# B&R Automation Studio project vibratorControlWithCurrentController (part 17)

```iecst
		0:
			IF this.responseStructMini.itemNo > 0 OR gMachineInterface.status.machineNotInProduction THEN // only start server when we are about to request images.
				brdkRESTServer_1.enable := TRUE;
				brdkRESTServer_1.pName := ADR('imageMini');
				brdkRESTServer_1.protocol := BRDK_REST_HTTP;
				brdkRESTServer_1.responseContentType := BRDK_REST_HTML;
				serverMini := 10;
			END_IF

		10:
			IF this.responseStructMini.image <> '' THEN
				brdkRESTServer_1.pResponseBody := ADR(this.responseStructMini.image);
				brdkRESTServer_1.responseBodyLength := SIZEOF(this.responseStructMini.image);
				brdkRESTServer_1.responseAction := BRDK_REST_200_OK;
			END_IF

			IF brdkRESTServer_1.status = ERR_OK THEN

			ELSIF brdkRESTServer_1.status <> ERR_FUB_BUSY THEN
				serverStatusError := brdkRESTServer_0.status;
				serverMini := 222;
			END_IF

		222:
			brdkRESTServer_1.enable := FALSE;
			this.TON_0.IN := TRUE;
			this.TON_0.PT := T#500ms;
			this.TON_0();

			IF this.TON_0.Q THEN
				this.TON_0.IN := FALSE;
				this.TON_0();

				serverMini := 0;
			END_IF

	END_CASE

	brdkRESTServer_1();

END_PROGRAM

PROGRAM _EXIT

	brdkRESTClient_0(enable := FALSE);
	brdkRESTServer_0(enable := FALSE);
END_PROGRAM
```

#### local.typ - Local data types
```iecst
TYPE
	local_typ : 	STRUCT
		strURL : STRING[300];
		oldItemNumber : STRING[20];
		errorCode : UINT;
		responeStruct : responeStruct_typ; (*JSON response will be parsed into this structure*)
		responseStructMini : responeStruct_typ;
		TON_0 : TON;
		imageURL : STRING[60];
		tmpStr : STRING[20];
		countPictureChanged : UDINT;
		tmpImageURL : STRING[60];
		TON_client : TON;
		errorCount : USINT;
	END_STRUCT;
	responeStruct_typ : 	STRUCT
		itemNo : DINT;
		image : STRING[99999];
	END_STRUCT;
END_TYPE
```

#### local.var - Local variables
```iecst
VAR
	brdkRESTClient_0 : brdkRESTClient;
	brdkRESTServer_0 : brdkRESTServer;
	requestBody : STRING[99];
	responseBody : STRING[99999];
	this : local_typ;
	state : USINT;
	serverState : USINT;
	message1 : DINT;
	message2 : DINT;
	pictureReady : BOOL;
	serverStatusError : UINT;
	strURL1 : STRING[80] := 'https://ip.uat.cz.pac.corp.lego.com/';
	strURL2 : STRING[80] := 'image-service/api/itemimage/getitemimagedata/';
	image : STRING[99999];
	testImg : USINT;
	oldTestImg : USINT;
	oldNumBricksInPortion : UDINT;
	item : STRING[80];
	quantity : STRING[99];
	serverMini : USINT;
	brdkRESTServer_1 : brdkRESTServer;
END_VAR
```

### Program Logical/services/EthernetIP/ethIp (IEC)

#### Variables.var
```iecst
VAR
	EIPInit_0 : EIPInit;
	EIPCyclic_0 : EIPCyclic;
	EIPExit_0 : EIPExit;
	remoteOutputArray : DINT;
	remoteInputArray : DINT;
	remoteCommectionStatus : UDINT;
	state : USINT;
	tmpStr : STRING[20];
	strInternalLineIP : STRING[20];
	ident : {REDUND_UNREPLICABLE} UDINT;
	ipLineController : STRING[15] := '192.168.1.10';
	interface : REFERENCE TO gEthernetIPInterface_typ;
END_VAR
```

#### Main.st
```iecst
PROGRAM _INIT

	EIPInit_0.enable := TRUE;
	EIPInit_0.pconfig := ADR('eipconf');
	EIPInit_0();

	remoteInputArray;
	remoteOutputArray;
	remoteCommectionStatus;
END_PROGRAM

PROGRAM _CYCLIC

	CASE state OF

		0:
			IF gMachineInterface.parameter.actualServerIP <> '' THEN

				tmpStr := '';
				brdkStrSubStr(ADR(tmpStr),ADR(gMachineInterface.parameter.actualServerIP),-1,3);
				strInternalLineIP := '192.168.1.';
				strInternalLineIP := CONCAT(strInternalLineIP,tmpStr);

				EIPCyclic_0.handle := EIPInit_0.handle;
				EIPCyclic_0.enable := TRUE;
				state := 10;
			END_IF

		10:
			interface ACCESS ADR(gEthernetIPInterface);

			remoteOutputArray.0  := interface.status.stop;
			remoteOutputArray.1  := interface.status.start;
			remoteOutputArray.2	 := interface.status.empty;
			remoteOutputArray.3  := interface.status.emptyMode;
			remoteOutputArray.4  := interface.status.bypassCassette;
			remoteOutputArray.13 := interface.status.di_cassetteReady;
			remoteOutputArray.14 := interface.status.di_cassetteQueue;
			remoteOutputArray.15 := interface.status.do_cassetteRelease;

			EIPCyclic_0();

			gMainInterface.cmd.stopEthIP := remoteInputArray.0;
			gMainInterface.cmd.startEthIP := remoteInputArray.1;
			gMainInterface.cmd.emptyEthIP := remoteInputArray.2;
			gMainInterface.cmd.emptyModeEthIP := remoteInputArray.3;
			gMainInterface.cmd.bypassCassetteEthIP := remoteInputArray.4;

	END_CASE

END_PROGRAM

PROGRAM _EXIT

	EIPExit_0.handle := EIPCyclic_0.handle;
	EIPExit_0.enable := TRUE;
	EIPExit_0();

END_PROGRAM
```

### Data object Logical/services/EthernetIP/eipconf (Simple)

#### DataObject.dat
```
"#OWNINTERFACE=SS1.IF1.ETH"
"#STATION=ROCKWELL"
"#STATIONIP=192.168.1.10"
"#STATIONSTATUS=::ethIp:remoteCommectionStatus"				; Number of active ethernet/IP connections.
"#CONNAME=EIPCon"
"#CONDIR=BOTH"
"#CONRPI=20"														; 20ms interval for requested packet. Need to call EIP FBs at least 2 times as fast as this time!
"#INPUTASSEMBLY=AssemIn"											; From AB side. This data is read by AB from B&R
"::ethIp:remoteOutputArray, DINT, 1"
"#OUTPUTASSEMBLY=AssemOut"											; From AB side. This data is read by B&R from AB
"::ethIp:remoteInputArray, DINT, 1"
```

### global.typ
```iecst
TYPE
	gEthernetIPInterface_typ : 	STRUCT
		status : gEthernetIPInterface_status_typ;
	END_STRUCT;
	gEthernetIPInterface_status_typ : 	STRUCT
		stop : BOOL; (*CM20 to LineController status*)
		start : BOOL; (*CM20 to LineController status*)
		empty : BOOL; (*CM20 to LineController status*)
		emptyMode : BOOL; (*CM20 to LineController status*)
		bypassCassette : BOOL; (*CM20 to LineController status*)
		di_cassetteReady : BOOL;
		di_cassetteQueue : BOOL;
		do_cassetteRelease : BOOL;
	END_STRUCT;
END_TYPE
```

### global.var
```iecst
VAR
	gEthernetIPInterface : gEthernetIPInterface_typ;
END_VAR
```

### dataGlobal.typ - Global data types
```iecst
TYPE
	gData_typ : 	STRUCT  (*Global recipe type.*)
		cmd : gData_cmd_typ; (*Command type.*)
		status : gData_status_typ; (*Status type.*)
	END_STRUCT;
	gData_cmd_typ : 	STRUCT  (*Global command type.*)
		numberOfSamples : UDINT := 250;
		triggerRecord : BOOL;
		exportRecord : BOOL;
		humanDecision : BOOL;
		machineDecision : BOOL;
		startRecord : BOOL;
		enable : BOOL;
	END_STRUCT;
	gData_status_typ : 	STRUCT  (*Global status type.*)
		running : BOOL := TRUE;
		active : BOOL;
		enoughFreeMem : BOOL; (*Will be false if we have less than 10 MiB freemem*)
	END_STRUCT;
END_TYPE
```

### dataGlobal.var - Global variables
```iecst
VAR
	gData : gData_typ; (*Global recipe interface.*)
END_VAR
```

### Package Logical/services/FAT - This module is used to handle all file devices.

### fatGlobal.typ - Global data types
```iecst
TYPE
	gFAT_typ : 	STRUCT  (*Global file type.*)
		cmd : gFAT_cmd_typ; (*File command type.*)
		status : gFAT_status_typ; (*File status type.*)
	END_STRUCT;
	gFAT_status_typ : 	STRUCT  (*File status type.*)
		dummy : BOOL; (*File devices are ready to use.*)
	END_STRUCT;
	gFAT_cmd_typ : 	STRUCT  (*File command type.*)
		dummy : BOOL; (*Update file devices command.*)
	END_STRUCT;
END_TYPE
```

### fatGlobal.var - Global variables
```iecst
VAR
	gFAT : gFAT_typ; (*Global file interface.*)
END_VAR
```

### Program Logical/services/FAT/FAT (IEC, version 1.00.0) - file device management task

#### local.st - Init, cyclic, exit code
```iecst
PROGRAM _INIT

	ST_name(0,ADR(this.configName),0);
	brdkStrCat(ADR(this.configName),ADR(':this.config'));
	ST_name(0,ADR(this.resultName),0);
	brdkStrCat(ADR(this.resultName),ADR(':resultFAT'));

	MpRecipeRegPar_Config.Enable := TRUE;
	this.MpRecipeXml_0.Load := TRUE;
	this.ton_chekForChanges.PT := T#5s;

END_PROGRAM

PROGRAM _CYCLIC

	// If machine aborts stop all tests.
	IF gMainInterface.status.state = STATE_ABORTED THEN
		this.hmi.testRunning88h := this.hmi.testRunning12h := FALSE;
	END_IF

	CASE state OF

		0:
			IF gFile.status.ready AND (gConfig.status.saved OR gConfig.status.loaded) AND this.resultsFATLoaded  THEN

				this.config.timeLeft88h := 88.0-(this.config.timeElapsed88h/3600);
				this.config.timeLeft88h := getHourMinutsFromDecimal(this.config.timeLeft88h);
				this.config.timeLeft12h := 12.0-(this.config.timeElapsed12h/3600);
				this.config.timeLeft12h := getHourMinutsFromDecimal(this.config.timeLeft12h);
				this.hmi.cmd.enableArrowNext := this.hmi.cmd.enableMenuNavigation := resultFAT.initialGroundMeas.done;

				state := 5;

			END_IF

		5:
			IF this.hmi.cmd.startFAT THEN
				// Only go to these states if FAT have been opened
				IF stateRetain > 0 THEN
					state := stateRetain;
				ELSE
					state := 10;
				END_IF
			END_IF

		10:
			// Initial ground measurements

			resultFAT.initialGroundMeas.firstMeasurementDone := resultFAT.initialGroundMeas.measurementValue <= 0.1 AND resultFAT.initialGroundMeas.measurementValue > 0.0;

			resultFAT.resistanceMeas2.done := TRUE;
			FOR i:=0 TO 9 DO

				CASE i OF

					0,1,2,3,7,8:	// 10ohm max resistance.
						IF resultFAT.resistanceMeas2.measurementArr[i]=0.0 OR resultFAT.resistanceMeas2.measurementArr[i] > 0.10 THEN
							resultFAT.resistanceMeas2.done := FALSE;
							resultFAT.resistanceMeas2.measurementOK[i] := FALSE;
						ELSE
							resultFAT.resistanceMeas2.measurementOK[i] := TRUE;
						END_IF

					4,5,6:		// 0.33ohm max resistance.
						IF resultFAT.resistanceMeas2.measurementArr[i]=0.0 OR resultFAT.resistanceMeas2.measurementArr[i] > 0.33 THEN
							resultFAT.resistanceMeas2.done := FALSE;
							resultFAT.resistanceMeas2.measurementOK[i] := FALSE;
						ELSE
							resultFAT.resistanceMeas2.measurementOK[i] := TRUE;
						END_IF

				END_CASE
			END_FOR

			resultFAT.initialGroundMeas.done := resultFAT.initialGroundMeas.firstMeasurementDone AND resultFAT.resistanceMeas2.done;

			this.hmi.cmd.enableArrowNext := this.hmi.cmd.enableMenuNavigation := resultFAT.initialGroundMeas.done;

			IF this.hmi.cmd.arrowNextValue THEN
				this.hmi.cmd.arrowNextValue := FALSE;
				IF resultFAT.initialGroundMeas.done THEN // only continue if it's done.
					state := 20;
				END_IF
			END_IF

		20:
			// Machine setup

			// On edgepos of input disable the oppsite (only 1 of 2 is valid)
			// A lot of information is depending on the machine type. All this information will be used at later steps in the FAT.
			IF EDGEPOS(this.hmi.cmd.smallCfToggleButton) THEN
				this.hmi.cmd.bigCfToggleButton := FALSE;
				gVibratorInterface[0].parameter.CFType := 0;
				gVibratorInterface[0].cmd.setCfType := TRUE;
				resultFAT.machineSetup.strCfSize := 'CM20 small';
				resultFAT.machineSetup.strMaxSpecsCF := 'MAX (2A/200V)';
				resultFAT.additionalInfo.weightOfCf := '5.5kg';
				resultFAT.CFSpringAdjust.strTargetFrequency := '48 - 51';
				resultFAT.CFCoilAdjust.magneticGap := 1.2;
				resultFAT.LFCoilAdjust.magneticGap := 0.6;
				resultFAT.machineSetup.cfSize := 0;
			ELSIF EDGEPOS(this.hmi.cmd.bigCfToggleButton) THEN
				this.hmi.cmd.smallCfToggleButton := FALSE;
				gVibratorInterface[0].parameter.CFType := 1;
				gVibratorInterface[0].cmd.setCfType := TRUE;
				resultFAT.machineSetup.strCfSize := 'CM20 large';
				resultFAT.machineSetup.strMaxSpecsCF := 'MAX (2A/200V)';
				resultFAT.additionalInfo.weightOfCf := '13.5kg';
				resultFAT.CFSpringAdjust.strTargetFrequency := '23.7 - 25.5';
				resultFAT.CFCoilAdjust.magneticGap := 2.5;
				resultFAT.LFCoilAdjust.magneticGap := 0.5;
				resultFAT.machineSetup.cfSize := 1;
			ELSIF EDGEPOS(this.hmi.cmd.leftDirectionOfRotation) THEN
				// direction should be 1 on left machine
				this.hmi.cmd.rightDirectionOfRotation := FALSE;
				gBeltInterface.cmd.setDirection := TRUE;
				gBeltInterface.parameter.direction := 1;
				resultFAT.machineSetup.strMachineType := 'Right';		// A machine with "left direction of rotation" is a right machine.
				resultFAT.machineSetup.strIsItALeftMachine := 'X (Left direction)';
				resultFAT.machineSetup.strIsItARightMachine := '';
				resultFAT.machineSetup.machineType := 0;	// left machine
				//config.machineType := 1;
			ELSIF EDGEPOS(this.hmi.cmd.rightDirectionOfRotation) THEN
				// direction should be 0 on right machine.
				this.hmi.cmd.leftDirectionOfRotation := FALSE;
				gBeltInterface.cmd.setDirection := TRUE;
				gBeltInterface.parameter.direction := 0;
				resultFAT.machineSetup.strMachineType := 'Left';		// A machine with "Right direction of rotation" is a left machine.
				resultFAT.machineSetup.strIsItALeftMachine := '';
				resultFAT.machineSetup.strIsItARightMachine := 'X (Right direction)';
				resultFAT.machineSetup.machineType := 1;	// right machine
				//config.machineType := 0;
			END_IF

			IF resultFAT.machineSetup.done THEN	// in order to load "this.hmi" if machine is restarted. They are not remanent.
				this.hmi.cmd.rightDirectionOfRotation := resultFAT.machineSetup.machineType=1;
				this.hmi.cmd.leftDirectionOfRotation := resultFAT.machineSetup.machineType=0;
				this.hmi.cmd.smallCfToggleButton := resultFAT.machineSetup.cfSize=0;
				this.hmi.cmd.bigCfToggleButton := resultFAT.machineSetup.cfSize=1;
			END_IF

			// Allow user to continue ONLY if their input is valid
			IF (this.hmi.cmd.smallCfToggleButton XOR this.hmi.cmd.bigCfToggleButton) AND
				(this.hmi.cmd.leftDirectionOfRotation XOR this.hmi.cmd.rightDirectionOfRotation) THEN
				resultFAT.machineSetup.done := TRUE;
				this.hmi.cmd.enableArrowNext := TRUE;
			ELSE
				resultFAT.machineSetup.done := FALSE;
				this.hmi.cmd.enableArrowNext := FALSE;
			END_IF

			// COMMENT OUT - this string anyways make 0 sense for report today?
//			IF EDGENEG(gVibratorInterface[0].cmd.setCfType) THEN	// a negative edge means it's done creating the string in vibrator task.
//				resultFAT.machineSetup.strLinearizationAccValuesCF := gVibratorInterface[0].status.strLinearizationAccValues;	// CF string
//				resultFAT.machineSetup.strLinearizationAccValuesLF := gVibratorInterface[1].status.strLinearizationAccValues;	// LF string
//			END_IF

			// User input to continue to next step
			IF this.hmi.cmd.arrowNextValue THEN
				this.hmi.cmd.arrowNextValue := FALSE;	// reset.

				// Set vibrator unit type and "top unit type" auto
				IF resultFAT.machineSetup.cfSize = 0 AND resultFAT.machineSetup.machineType = 0 THEN	//  small and left
					resultFAT.additionalInfo.vibratorUnitType := 'SRC-N 250-2L-LEGO II';
					resultFAT.additionalInfo.topUnitType := 'PJ 2016 HA';
				ELSIF resultFAT.machineSetup.cfSize = 0 AND resultFAT.machineSetup.machineType = 1 THEN	//  small and right
					resultFAT.additionalInfo.vibratorUnitType := 'SRC-N 250-2R-LEGO II';
					resultFAT.additionalInfo.topUnitType := 'PJ 2016 VA';
				ELSIF resultFAT.machineSetup.cfSize = 1 AND resultFAT.machineSetup.machineType = 0 THEN	//  big and left
					resultFAT.additionalInfo.vibratorUnitType := 'SRC-N 400-1L-LEGO III';
					resultFAT.additionalInfo.topUnitType := 'PJ 99 HA';
				ELSIF resultFAT.machineSetup.cfSize = 1 AND resultFAT.machineSetup.machineType = 1 THEN	//  big and right
					resultFAT.additionalInfo.vibratorUnitType := 'SRC-N 400-1R-LEGO III';
					resultFAT.additionalInfo.topUnitType := 'PJ 99 VA';
				END_IF

				state := 30;
			ELSIF this.hmi.cmd.arrowBackValue THEN
				this.hmi.cmd.arrowBackValue := FALSE;
				state := 10;
			END_IF

		30:
			// Wing connector (wingTestIO)

			IF this.hmi.cmd.arrowNextValue THEN			// go to next
				this.hmi.cmd.arrowNextValue := FALSE;	// reset
				state := 40;
			ELSIF this.hmi.cmd.arrowBackValue THEN
				this.hmi.cmd.arrowBackValue := FALSE;
				state := 20;
			END_IF

		40:
			// Additional machine info

			// Create string typeNo.-SerialNo.
			IF resultFAT.additionalInfo.serialNo <> '' AND resultFAT.additionalInfo.typeNo <> '' THEN
				brdkStrMemSet(ADR(resultFAT.additionalInfo.typeNoAndSerialNo),0,SIZEOF(resultFAT.additionalInfo.typeNoAndSerialNo));
				brdkStrCat(ADR(resultFAT.additionalInfo.typeNoAndSerialNo),ADR(resultFAT.additionalInfo.typeNo));
				this.tmpString := '-';
				brdkStrCat(ADR(resultFAT.additionalInfo.typeNoAndSerialNo),ADR(this.tmpString));
				brdkStrCat(ADR(resultFAT.additionalInfo.typeNoAndSerialNo),ADR(resultFAT.additionalInfo.serialNo));

				// SerialNoDINT
				this.tmpString := '';
				brdkStrCat(ADR(this.tmpString),ADR(resultFAT.additionalInfo.typeNo));
				brdkStrCat(ADR(this.tmpString),ADR(resultFAT.additionalInfo.serialNo));
				gMachineInterface.cmd.serialNoDINT := STRING_TO_DINT(this.tmpString); //interface.par.serialNoDINT := STRING_TO_DINT(this.tmpString);
			END_IF
			//interface.par.serialNo := resultFAT.additionalInfo.typeNoAndSerialNo;

			// Load "this.hmi.status" texts if they are empty and resultFAT is not (Happens on a warm restart).
			IF this.hmi.status.additionalInfo.typeNo = 0 AND resultFAT.additionalInfo.typeNo <> '' THEN
				this.hmi.status.additionalInfo.typeNo := STRING_TO_UDINT(resultFAT.additionalInfo.typeNo);
			END_IF
			IF this.hmi.status.additionalInfo.serialNo = 0 AND resultFAT.additionalInfo.serialNo <> '' THEN
				this.hmi.status.additionalInfo.serialNo := STRING_TO_UDINT(resultFAT.additionalInfo.serialNo);
			END_IF
			IF this.hmi.status.additionalInfo.rnoNo = 0.0 AND resultFAT.additionalInfo.rnaProductNo <> '' THEN
				this.hmi.status.additionalInfo.rnoNo := STRING_TO_LREAL(resultFAT.additionalInfo.rnaProductNo);
			END_IF
			IF this.hmi.status.additionalInfo.topSerialNo = 0 AND resultFAT.additionalInfo.topSerialNo <> '' THEN
				this.hmi.status.additionalInfo.topSerialNo := STRING_TO_UDINT(resultFAT.additionalInfo.topSerialNo);
			END_IF

			// Put int into strings for report
			resultFAT.additionalInfo.typeNo := UDINT_TO_STRING(this.hmi.status.additionalInfo.typeNo);
			resultFAT.additionalInfo.serialNo := UDINT_TO_STRING(this.hmi.status.additionalInfo.serialNo);
			resultFAT.additionalInfo.rnaProductNo := LREAL_TO_STRING(this.hmi.status.additionalInfo.rnoNo);
			resultFAT.additionalInfo.topSerialNo := UDINT_TO_STRING(this.hmi.status.additionalInfo.topSerialNo);

			IF this.hmi.status.additionalInfo.IRTHno <> this.oldLREAL THEN
				resultFAT.additionalInfo.IRTHno := LREAL_TO_STRING(this.hmi.status.additionalInfo.IRTHno);
				brdkStrRemove(ADR(resultFAT.additionalInfo.IRTHno),(brdkStrLen(ADR(resultFAT.additionalInfo.IRTHno))-2),2);

				IF this.hmi.status.additionalInfo.IRTHno>10000000 THEN // hacky way to append a space to a numeric input from HMI.
					this.tmpString := ' ';
					brdkStrInsertAtPos(ADR(resultFAT.additionalInfo.IRTHno),ADR(this.tmpString),6);
				END_IF
			END_IF
			this.oldLREAL := this.hmi.status.additionalInfo.IRTHno;

			IF this.hmi.cmd.arrowNextValue THEN
				this.hmi.cmd.arrowNextValue := FALSE;
				state := 50;
			ELSIF this.hmi.cmd.arrowBackValue THEN
				this.hmi.cmd.arrowBackValue := FALSE;
				state := 30;
			END_IF

			// If some chars in all text inputs the test is done:
			IF resultFAT.additionalInfo.IRTHno <> '0' AND resultFAT.additionalInfo.IRTHno <> '0.0' AND resultFAT.additionalInfo.rnaProductNo <> '0.0' AND resultFAT.additionalInfo.typeNo <> '0' AND resultFAT.additionalInfo.serialNo <> '0' AND resultFAT.additionalInfo.topSerialNo <> '0' AND resultFAT.additionalInfo.topUnitType <> '' AND resultFAT.additionalInfo.vibratorUnitType <> '' THEN
				resultFAT.additionalInfo.done := TRUE;
			ELSE
				resultFAT.additionalInfo.done := FALSE;
			END_IF

		50:

			//Capcon voltage measurement

			// Check if user input is in the expected interval
			IF resultFAT.capconMeasurement.V1 >= 18 - this.maxPlusMinusVoltage AND resultFAT.capconMeasurement.V1 <= 18 + this.maxPlusMinusVoltage THEN
				this.hmi.cmd.crossmarkV1 := 1;
			ELSE
				this.hmi.cmd.crossmarkV1 := 0;
			END_IF

			// Check if user input is in the expected interval
			IF resultFAT.capconMeasurement.V2 >= -15.8 - this.maxPlusMinusVoltage AND resultFAT.capconMeasurement.V2 <= -15.8 + this.maxPlusMinusVoltage THEN
				this.hmi.cmd.crossmarkV2 := 1;
			ELSE
				this.hmi.cmd.crossmarkV2 := 0;
			END_IF

			IF (this.hmi.cmd.crossmarkV1 > 0 AND this.hmi.cmd.crossmarkV2 > 0) THEN
				resultFAT.capconMeasurement.done := TRUE;
				this.hmi.cmd.enableArrowNext := TRUE;
			ELSE
				resultFAT.capconMeasurement.done := FALSE;
				this.hmi.cmd.enableArrowNext := FALSE;
			END_IF

			IF this.hmi.cmd.arrowNextValue THEN
				this.hmi.cmd.arrowNextValue := FALSE;
				state := 60;
			ELSIF this.hmi.cmd.arrowBackValue THEN
				this.hmi.cmd.arrowBackValue := FALSE;
				state := 40;
			END_IF

		60:
			//	em.description := 'Capcon signal test';
			// 1st test. Test that an analog input is getting into the machine when dropping something through capcon:

			// 2nd test. Auto test MAX speed signal doing a period of 5s.
			IF EDGEPOS(this.hmi.cmd.startCapconTest2) THEN
				gCapconInterface.status.maxRawSignal := 0;
				gCapconInterface.cmd.startSpeedSignalTest := TRUE;
			END_IF

			IF EDGENEG(gCapconInterface.cmd.startSpeedSignalTest) THEN
				this.hmi.cmd.startCapconTest2 := FALSE;
				this.hmi.status.maxRawSignal := ABS(gCapconInterface.status.maxRawSignal);
				IF this.hmi.status.maxRawSignal>1 AND ABS(this.hmi.status.maxRawSignal) < 100 THEN // TODO: 40 NEEDS TO BE TESTED!
					resultFAT.capconTest.signalTest2 := TRUE;
				ELSE
					resultFAT.capconTest.signalTest2 := FALSE;
				END_IF
			END_IF

			IF this.hmi.cmd.arrowNextValue THEN
				this.hmi.cmd.arrowNextValue := FALSE;
				state := 70;
			ELSIF this.hmi.cmd.arrowBackValue THEN
				this.hmi.cmd.arrowBackValue := FALSE;
				state := 50;
			END_IF

			resultFAT.capconTest.done := resultFAT.capconTest.signalTest1 AND resultFAT.capconTest.signalTest2;

		70:
			// em.description := 'Level sensor test';

			gFeederInterface.cmd.levelSensorTestActive := TRUE;

			IF this.hmi.cmd.doLevelSensorTest AND resultFAT.levelSensorTest.receiverOK THEN

				// level sensor test.
				CASE levelTestState OF

					0:
						gFeederInterface.cmd.setLevelSensor[0] := FALSE;
						gFeederInterface.cmd.setLevelSensor[1] := FALSE;
						gFeederInterface.cmd.setLevelSensor[2] := TRUE;
						resultFAT.levelSensorTest.transmitterLowOK := FALSE;
						resultFAT.levelSensorTest.transmitterMediumOK := FALSE;
						resultFAT.levelSensorTest.transmitterHighOK := FALSE;
						resultFAT.levelSensorTest.operatorApproveLow := resultFAT.levelSensorTest.operatorApproveMedium := resultFAT.levelSensorTest.operatorApproveHigh := FALSE;

						this.timeElapsed := 0;
						levelTestState := 5;

					5:	// wait 1s
						this.timeElapsed := this.timeElapsed + 40000;
						IF this.timeElapsed > 1000000 THEN
							this.timeElapsed := 0;
							IF gFeederInterface.status.levelSensorReceiverInBowl THEN
								levelTestState := 222;
							ELSE
								this.hmi.status.styleToggleInputHigh := TRUE;
								levelTestState := 10;
							END_IF
						END_IF

					10: // Wait for user to approve that HIGH transmitter is flashing.

						IF gFeederInterface.status.levelSensorReceiverInBowl THEN
							levelTestState := 222;
						ELSIF resultFAT.levelSensorTest.operatorApproveHigh THEN
							resultFAT.levelSensorTest.transmitterHighOK := TRUE;

							gFeederInterface.cmd.setLevelSensor[0] := FALSE;
							gFeederInterface.cmd.setLevelSensor[1] := TRUE;
							gFeederInterface.cmd.setLevelSensor[2] := FALSE;
							this.hmi.status.styleToggleInputHigh := FALSE;
							this.hmi.status.styleToggleInputMedium := TRUE;
							levelTestState := 20;
						END_IF

					20: // Wait for user to approve that MEDIUM transmitter is flashing.

						IF gFeederInterface.status.levelSensorReceiverInBowl THEN
							levelTestState := 222;
						ELSIF resultFAT.levelSensorTest.operatorApproveMedium THEN
							resultFAT.levelSensorTest.transmitterMediumOK := TRUE;

							gFeederInterface.cmd.setLevelSensor[0] := TRUE;
							gFeederInterface.cmd.setLevelSensor[1] := FALSE;
							gFeederInterface.cmd.setLevelSensor[2] := FALSE;
							this.hmi.status.styleToggleInputMedium := FALSE;
							this.hmi.status.styleToggleInputLow := TRUE;

							levelTestState := 30;
						END_IF

					30: //  Wait for user to approve that LOW transmitter is flashing.

						IF gFeederInterface.status.levelSensorReceiverInBowl THEN
							levelTestState := 222;
						ELSIF resultFAT.levelSensorTest.operatorApproveLow THEN
							resultFAT.levelSensorTest.transmitterLowOK := TRUE;

							gFeederInterface.cmd.setLevelSensor[0] := FALSE;
							gFeederInterface.cmd.setLevelSensor[1] := FALSE;
							gFeederInterface.cmd.setLevelSensor[2] := FALSE;
							this.hmi.status.styleToggleInputLow := FALSE;
							this.hmi.cmd.doLevelSensorTest := FALSE;
							levelTestState := 0;
						END_IF

					222:
						//test failed reset everything
						this.hmi.cmd.doLevelSensorTest := FALSE;
						gFeederInterface.cmd.setLevelSensor[0] := FALSE;
						gFeederInterface.cmd.setLevelSensor[1] := FALSE;
						gFeederInterface.cmd.setLevelSensor[2] := FALSE;
						resultFAT.levelSensorTest.operatorApproveHigh := resultFAT.levelSensorTest.operatorApproveMedium := resultFAT.levelSensorTest.operatorApproveLow := FALSE;
						resultFAT.levelSensorTest.transmitterLowOK := FALSE;
						resultFAT.levelSensorTest.transmitterMediumOK := FALSE;
						resultFAT.levelSensorTest.transmitterHighOK := FALSE;
						this.hmi.status.styleToggleInputHigh := this.hmi.status.styleToggleInputMedium := this.hmi.status.styleToggleInputLow := FALSE;
						levelTestState := 0;

				END_CASE

			ELSIF this.hmi.cmd.doLevelSensorTest THEN
				this.hmi.cmd.doLevelSensorTest := FALSE; // reset if user presses button when receiver is not OK.
			ELSE
				// manuel control from user.
				gFeederInterface.cmd.setLevelSensor[0] := this.hmi.cmd.setLevelSensorLow;
				gFeederInterface.cmd.setLevelSensor[1] := this.hmi.cmd.setLevelSensorMedium;
				gFeederInterface.cmd.setLevelSensor[2] := this.hmi.cmd.setLevelSensorHigh;

				IF NOT this.hmi.cmd.setLevelSensorHigh AND NOT this.hmi.cmd.setLevelSensorMedium AND NOT this.hmi.cmd.setLevelSensorLow THEN
					// if receiver is high when all transmitters are low the receiver is OK.
					IF gFeederInterface.status.levelSensorReceiverInBowl THEN
						resultFAT.levelSensorTest.receiverOK := TRUE;
					ELSE
						resultFAT.levelSensorTest.receiverOK := FALSE;
					END_IF
				END_IF

			END_IF

			IF this.hmi.cmd.arrowNextValue THEN
				this.hmi.cmd.arrowNextValue := FALSE;	// reset.
				gFeederInterface.cmd.levelSensorTestActive := FALSE;
				state := 80;
			ELSIF this.hmi.cmd.arrowBackValue THEN
				this.hmi.cmd.arrowBackValue := FALSE;
				gFeederInterface.cmd.levelSensorTestActive := FALSE;
				state := 60;
			END_IF

			resultFAT.levelSensorTest.done := resultFAT.levelSensorTest.receiverOK AND resultFAT.levelSensorTest.transmitterHighOK AND resultFAT.levelSensorTest.transmitterMediumOK AND resultFAT.levelSensorTest.transmitterLowOK;
			//this.hmi.cmd.enableArrowNext := resultFAT.levelSensorTest.done;

		80:
			//  'Photo sensor adjustment';

			IF this.hmi.cmd.arrowNextValue THEN
				this.hmi.cmd.arrowNextValue := FALSE;	// reset.
				state := 90;
			ELSIF this.hmi.cmd.arrowBackValue THEN
				this.hmi.cmd.arrowBackValue := FALSE;
				state := 70;
			END_IF

			this.hmi.cmd.enableArrowNext := resultFAT.photoSensorAdjust.done;

		90:
		//	em.description := 'Wait for automatic test of photo sensor to be done';

			IF EDGEPOS(this.hmi.cmd.doPhotoSensorTest) THEN		// Start the test.

				this.hmi.status.photoSensorTestText := 0;
				gBeltInterface.cmd.doPhotoSensorTest := TRUE;						// signal to belt that it should start automatic test.
			ELSIF EDGEPOS(this.hmi.cmd.doPhotoSensorTestNoBelt) THEN

				gBeltInterface.cmd.doPhotoSensorTestNoBelt := TRUE;
			ELSE
				IF gBeltInterface.status.photoSensorTestResult = TEST_STOPPED THEN
					resultFAT.photoSensorTest.testWithBelt := FALSE;
					gBeltInterface.status.photoSensorTestResult := TEST_NOT_DONE;
					this.hmi.cmd.doPhotoSensorTest := FALSE;
					this.hmi.status.photoSensorTestText := 3;	// test stopped text
				ELSIF gBeltInterface.status.photoSensorTestResult = TEST_NOT_OK THEN	// Something went wrong doing test.
					resultFAT.photoSensorTest.testWithBelt := FALSE;
					gBeltInterface.status.photoSensorTestResult := TEST_NOT_DONE;
					this.hmi.cmd.doPhotoSensorTest := FALSE;
					this.hmi.status.photoSensorTestText := 2;
				ELSIF gBeltInterface.status.photoSensorTestResult = TEST_OK THEN
					resultFAT.photoSensorTest.testWithBelt := TRUE;
					gBeltInterface.status.photoSensorTestResult := TEST_NOT_DONE;
					this.hmi.cmd.doPhotoSensorTest := FALSE;
					this.hmi.status.photoSensorTestText := 1;
				END_IF

				IF gBeltInterface.status.photoSensorTestNoBeltResult = TEST_STOPPED THEN
					resultFAT.photoSensorTest.testWithNoBelt := FALSE;
					gBeltInterface.status.photoSensorTestNoBeltResult := TEST_NOT_DONE;
					this.hmi.cmd.doPhotoSensorTestNoBelt := FALSE;
				ELSIF gBeltInterface.status.photoSensorTestNoBeltResult = TEST_NOT_OK THEN	// Something went wrong doing test.
					resultFAT.photoSensorTest.testWithNoBelt := FALSE;
					gBeltInterface.status.photoSensorTestNoBeltResult := TEST_NOT_DONE;
					this.hmi.cmd.doPhotoSensorTestNoBelt := FALSE;
				ELSIF gBeltInterface.status.photoSensorTestNoBeltResult = TEST_OK THEN
					resultFAT.photoSensorTest.testWithNoBelt := TRUE;
					gBeltInterface.status.photoSensorTestNoBeltResult := TEST_NOT_DONE;
					this.hmi.cmd.doPhotoSensorTestNoBelt := FALSE;
				END_IF

			END_IF

			IF this.hmi.cmd.arrowNextValue THEN			// go to next
				this.hmi.cmd.arrowNextValue := FALSE;	// reset
				state := 100;
			ELSIF this.hmi.cmd.arrowBackValue THEN
				this.hmi.cmd.arrowBackValue := FALSE;
				state := 80;
			END_IF

			IF resultFAT.photoSensorTest.testWithBelt THEN
				this.hmi.status.photoSensorTestText := 1;
			END_IF
			resultFAT.photoSensorTest.done := resultFAT.photoSensorTest.testWithBelt AND resultFAT.photoSensorTest.testWithNoBelt;
			this.hmi.cmd.enableArrowNext := resultFAT.photoSensorTest.done;

		100:
			// 'Belt feeder test IO - 1';

			IF EDGEPOS(this.hmi.cmd.doBfFlapTest) THEN
				//	this.hmi.cmd.doBfFlapTest := FALSE;		// reset this when test is done instead!!
				// start flap test in feeder task
				resultFAT.bfTestIO.flapTestDone := FALSE;
				gFeederInterface.cmd.startFlapTest := TRUE;
			ELSE
				// reach on test result from flap test.
				IF gFeederInterface.status.flapTest = TEST_STOPPED THEN
					resultFAT.bfTestIO.flapTestDone := FALSE;
					gFeederInterface.status.flapTest := TEST_NOT_DONE;
					this.hmi.cmd.doBfFlapTest := FALSE;
				ELSIF gFeederInterface.status.flapTest = TEST_NOT_OK THEN	// Something went wrong doing test.
					resultFAT.bfTestIO.flapTestDone := FALSE;
					gFeederInterface.status.flapTest := TEST_NOT_DONE;
					this.hmi.cmd.doBfFlapTest := FALSE;
				ELSIF gFeederInterface.status.flapTest = TEST_OK THEN
					resultFAT.bfTestIO.flapTestDone := TRUE;
					gFeederInterface.status.flapTest := TEST_NOT_DONE;
					this.hmi.cmd.doBfFlapTest := FALSE;
				END_IF
			END_IF

			resultFAT.bfTestIO.done := resultFAT.bfTestIO.approveIOsManually AND resultFAT.bfTestIO.approveMainsVoltage AND resultFAT.bfTestIO.flapTestDone;

			IF this.hmi.cmd.arrowNextValue THEN			// go to next
				this.hmi.cmd.arrowNextValue := FALSE;	// reset
				state := 110;
			ELSIF this.hmi.cmd.arrowBackValue THEN
				this.hmi.cmd.arrowBackValue := FALSE;
				state := 90;
			END_IF

		110:
			// 'Wing test IO - flap namur sensor, cassette signal, dosing signal, cassette queue';

			IF EDGEPOS(this.hmi.cmd.doWingTestManuel) THEN
				//this.hmi.cmd.doWingTestManuel := FALSE;
				gUpperFlapInterface.cmd.wingTestManual := TRUE; // Only start upper - they will start each other "sequantially"

				// Reset test results
				resultFAT.wingTestIO.upperFlapOK := FALSE;
				resultFAT.wingTestIO.middleFlapOK := FALSE;
				resultFAT.wingTestIO.bottomFlapOK := FALSE;
				resultFAT.wingTestIO.neighbourFlapOK := FALSE;
				resultFAT.wingTestIO.cassetteReleaseOK := FALSE;
				resultFAT.wingTestIO.ioTestOK := FALSE;

			END_IF

			IF this.hmi.cmd.doWingTestManuel THEN

				// Wait for all tests to be done
				IF NOT gUpperFlapInterface.cmd.wingTestManual AND NOT gMiddleFlapInterface.cmd.wingTestManual AND NOT gBottomFlapInterface.cmd.wingTestManual AND NOT gCassetteInterface.cmd.wingTestManual THEN
					this.hmi.cmd.doWingTestManuel := FALSE;

					// write result from test into resultFAT struct
					resultFAT.wingTestIO.upperFlapOK := gUpperFlapInterface.status.testResultFAT;
					resultFAT.wingTestIO.middleFlapOK := gMiddleFlapInterface.status.testResultFAT;
					resultFAT.wingTestIO.bottomFlapOK := gBottomFlapInterface.status.testResultFAT;
					resultFAT.wingTestIO.neighbourFlapOK := gBottomFlapInterface.status.testResultFAT; // bottom also test neighbour
					resultFAT.wingTestIO.cassetteReleaseOK := gCassetteInterface.status.testResultFAT;
					resultFAT.wingTestIO.ioTestOK := resultFAT.wingTestIO.upperFlapOK AND resultFAT.wingTestIO.middleFlapOK AND resultFAT.wingTestIO.bottomFlapOK AND resultFAT.wingTestIO.neighbourFlapOK AND resultFAT.wingTestIO.cassetteReleaseOK;

				END_IF

			END_IF

			resultFAT.wingTestIO.done := resultFAT.wingTestIO.ioTestOK AND resultFAT.wingTestIO.approveFunctionality;

			IF this.hmi.cmd.arrowNextValue THEN			// go to next
				this.hmi.cmd.arrowNextValue := FALSE;	// reset
				state := 120;
			ELSIF this.hmi.cmd.arrowBackValue THEN
				this.hmi.cmd.arrowBackValue := FALSE;
				state := 100;
			END_IF

		120:
			//	'CF coils adjustments';

			this.hmi.status.isSmallMachine := gVibratorInterface[0].parameter.machineSize=0;
			this.hmi.status.isBigMachine := gVibratorInterface[0].parameter.machineSize=1;

			IF this.hmi.cmd.arrowNextValue THEN
				this.hmi.cmd.arrowNextValue := FALSE;	// reset.
				// Set default amount of plates if all plate values are set to 0 (means no user input).
				FOR i:=0 TO 2 DO
					IF resultFAT.CFSpringAdjust.plate08mm[i] > 0 OR resultFAT.CFSpringAdjust.plate09mm[i] > 0 OR resultFAT.CFSpringAdjust.plate15mm[i] > 0 OR resultFAT.CFSpringAdjust.plate20mm[i] > 0 OR resultFAT.CFSpringAdjust.plate25mm[i] > 0 THEN
						EXIT;
					ELSIF i=2 THEN	// If all all values are 0 set the default amount of plates for this CF.
						IF resultFAT.machineSetup.cfSize=0 THEN // Default for small cf is 5 2.0mm plates on each spring.
							resultFAT.CFSpringAdjust.plate20mm[0] := 5;
							resultFAT.CFSpringAdjust.plate20mm[1] := 5;
							resultFAT.CFSpringAdjust.plate20mm[2] := 5;
						ELSE	// default for big cf is 7 2.0mm plates on each spring
							resultFAT.CFSpringAdjust.plate20mm[0] := 7;
							resultFAT.CFSpringAdjust.plate20mm[1] := 7;
							resultFAT.CFSpringAdjust.plate20mm[2] := 7;
						END_IF
					END_IF

				END_FOR

				state := 130;
			ELSIF this.hmi.cmd.arrowBackValue THEN
				this.hmi.cmd.arrowBackValue := FALSE;
				state := 110;
			END_IF

		130:
			// CF spring adjustments

			IF this.hmi.cmd.startCalibration THEN
				this.hmi.cmd.startCalibration := FALSE;
				// Need to use this bool to differentiate if it was a "FAT calibration" or a "normal calibration".
				gVibratorInterface[0].status.calibratingMode := TRUE;
				this.cfCali := TRUE;
			END_IF

			IF gVibratorInterface[0].status.calibrationResultsReady THEN
				gVibratorInterface[0].status.calibrationResultsReady := FALSE;
				this.hmi.cmd.startCalibration := FALSE;

				IF this.cfCali THEN
					// Take results from calibration and save in resultFAT
					resultFAT.CFSpringAdjust.ressFrequency := gVibratorInterface[0].status.calibrationResultFrequency;
					resultFAT.CFSpringAdjust.maxCurrent := gVibratorInterface[0].status.calibrationResultCurrent;
					resultFAT.CFSpringAdjust.currentOK := gVibratorInterface[0].status.calibrationResultCurrentOK;
					resultFAT.CFSpringAdjust.frequencyOK := gVibratorInterface[0].status.calibrationResultFrequencyOK;
				END_IF
				this.cfCali := FALSE;
			END_IF

			resultFAT.CFSpringAdjust.done := resultFAT.CFSpringAdjust.currentOK AND resultFAT.CFSpringAdjust.frequencyOK;

			IF this.hmi.cmd.arrowNextValue THEN			// go to next
				this.hmi.cmd.arrowNextValue := FALSE;	// reset
				state := 140;
			ELSIF this.hmi.cmd.arrowBackValue THEN
				this.hmi.cmd.arrowBackValue := FALSE;
				state := 120;
			END_IF

		140:
			// 'LF coils adjustment';	// might need to make more substates for CF and LF.

			IF this.hmi.cmd.arrowNextValue THEN
				this.hmi.cmd.arrowNextValue := FALSE;	// reset.
				// Set default amount of plates if all plate values are set to 0 (means no user input).
				FOR i:=0 TO 1 DO
					IF resultFAT.LFSpringAdjust.plate08mm[i] > 0 OR resultFAT.LFSpringAdjust.plate09mm[i] > 0 OR resultFAT.LFSpringAdjust.plate15mm[i] > 0 OR resultFAT.LFSpringAdjust.plate20mm[i] > 0 OR resultFAT.LFSpringAdjust.plate25mm[i] > 0 THEN
						EXIT;
					ELSIF i=1 THEN	// If all all values are 0 set the default amount of plates for this CF.
						IF resultFAT.machineSetup.cfSize=0 THEN // Default for small cm
							resultFAT.LFSpringAdjust.plate08mm[0] := 2;
							resultFAT.LFSpringAdjust.plate08mm[1] := 1;
						ELSE	// default for big cm
							resultFAT.LFSpringAdjust.plate08mm[0] := 1;
							resultFAT.LFSpringAdjust.plate08mm[1] := 1;
							resultFAT.LFSpringAdjust.plate09mm[0] := 1;
						END_IF
					END_IF

				END_FOR

				state := 150;
			ELSIF this.hmi.cmd.arrowBackValue THEN
				this.hmi.cmd.arrowBackValue := FALSE;
				state := 130;
			END_IF

		150:
			// LF calibration

			IF this.hmi.cmd.startCalibration THEN
				this.hmi.cmd.startCalibration := FALSE;
				// Need to use this bool to differentiate if it was a "FAT calibration" or a "normal calibration".
				gVibratorInterface[1].status.calibratingMode := TRUE;
				this.lfCali := TRUE;
			END_IF

			IF gVibratorInterface[1].status.calibrationResultsReady THEN
				gVibratorInterface[1].status.calibrationResultsReady := FALSE;
				this.hmi.cmd.startCalibration := FALSE;

				IF this.lfCali THEN
					// Take results from calibration and save in resultFAT
					resultFAT.LFSpringAdjust.ressFrequency := gVibratorInterface[1].status.calibrationResultFrequency;
					resultFAT.LFSpringAdjust.maxCurrent := gVibratorInterface[1].status.calibrationResultCurrent;
					resultFAT.LFSpringAdjust.currentOK := gVibratorInterface[1].status.calibrationResultCurrentOK;
					resultFAT.LFSpringAdjust.frequencyOK := gVibratorInterface[1].status.calibrationResultFrequencyOK;

					resultFAT.LFSpringAdjust.strResultForReport := REAL_TO_STRING(resultFAT.LFSpringAdjust.maxCurrent);
					resultFAT.LFSpringAdjust.strResultForReport := CONCAT(resultFAT.LFSpringAdjust.strResultForReport,'A');
					resultFAT.LFSpringAdjust.strResultForReport := CONCAT(resultFAT.LFSpringAdjust.strResultForReport,' / ');
					this.tmpString := REAL_TO_STRING(resultFAT.LFSpringAdjust.ressFrequency);
					resultFAT.LFSpringAdjust.strResultForReport := CONCAT(resultFAT.LFSpringAdjust.strResultForReport,this.tmpString);
					resultFAT.LFSpringAdjust.strResultForReport := CONCAT(resultFAT.LFSpringAdjust.strResultForReport,'Hz');

				END_IF
				this.lfCali := FALSE;
			END_IF

			resultFAT.LFSpringAdjust.done := resultFAT.LFSpringAdjust.currentOK AND resultFAT.LFSpringAdjust.frequencyOK;

			IF this.hmi.cmd.arrowNextValue THEN			// go to next
				this.hmi.cmd.arrowNextValue := FALSE;	// reset
				state := 160;
			ELSIF this.hmi.cmd.arrowBackValue THEN
				this.hmi.cmd.arrowBackValue := FALSE;
				state := 140;
			END_IF

		160:
			// 88h test
			this.testRunning := this.hmi.testRunning88h XOR this.hmi.testRunning12h;
			gBeltInterface.cmd.runManualTest := gVibratorInterface[0].cmd.runManualTest := gVibratorInterface[1].cmd.runManualTest := this.testRunning;

			IF this.hmi.testRunning88h AND this.hmi.testRunning12h THEN
				// Both can't run at the same time. Disable both if user tries to do this.
				this.hmi.testRunning88h := this.hmi.testRunning12h := FALSE;
			ELSIF this.hmi.testRunning88h THEN

				// Start belt and vibrators
				gBeltInterface.parameter.speedManualTest := 400.0;
				gVibratorInterface[0].parameter.speedPctManualTest := SEL(this.config.timeElapsed88h > 43200,40.0,80.0); // First 12h use 40% rest of the time use 80% (43200s = 12hours)
				gVibratorInterface[1].parameter.speedPctManualTest := 100.0;

				// Calculate time
				this.config.timeElapsed88h := this.config.timeElapsed88h + CYCLE_TIME_seconds;
				this.config.timeLeft88h := 88.0-(this.config.timeElapsed88h/3600);
				this.config.timeLeft88h := getHourMinutsFromDecimal(this.config.timeLeft88h);

				IF this.config.timeLeft88h <= 0.0 THEN
					this.hmi.testRunning88h := this.hmi.testRunning12h := FALSE;
					gConfig.cmd.save := TRUE;
					this.config.timeLeft88h := 0.0;
					resultFAT.longTest88h.done := TRUE;
				END_IF

			END_IF

			// Save to config every 10min
			this.TON_0.IN := this.testRunning;
			this.TON_0.PT := T#10m;
			this.TON_0();

			IF this.TON_0.Q THEN
				this.TON_0.IN := FALSE;
				this.TON_0();

				gConfig.cmd.save := TRUE;
			END_IF

			// If test not running set parameter to 0.
			IF NOT this.testRunning THEN
				gVibratorInterface[0].parameter.speedPctManualTest := 0.0;
				gVibratorInterface[1].parameter.speedPctManualTest := 0.0;
			END_IF

			IF this.hmi.cmd.arrowNextValue THEN			// go to next
				this.hmi.cmd.arrowNextValue := FALSE;	// reset
				state := 170;
			ELSIF this.hmi.cmd.arrowBackValue THEN
				this.hmi.cmd.arrowBackValue := FALSE;
				state := 150;
			END_IF

		170:
			// 'After 72H test adjustments';

			resultFAT.after72hAdjustments.done := resultFAT.after72hAdjustments.approveCoverMounting AND resultFAT.after72hAdjustments.approveHabasitMounting AND resultFAT.after72hAdjustments.approvePacemakerMarking AND resultFAT.after72hAdjustments.approveRNAmarking;

			IF this.hmi.cmd.arrowNextValue THEN
				this.hmi.cmd.arrowNextValue := FALSE;	// reset.
				state := 180;
			ELSIF this.hmi.cmd.arrowBackValue THEN
				this.hmi.cmd.arrowBackValue := FALSE;
				state := 160;
			END_IF

		180:
			// Calibrate CF again after habasit (LF should not be needed since it has habasit on from the start)

			IF this.hmi.cmd.startCalibration THEN
				this.hmi.cmd.startCalibration := FALSE;
				this.cfCaliHabasit := TRUE; //save what kind of FAT cali which is running.
				gVibratorInterface[0].status.calibratingMode := TRUE;
			END_IF

			IF gVibratorInterface[0].status.calibrationResultsReady THEN
				gVibratorInterface[0].status.calibrationResultsReady := FALSE;

				IF this.cfCaliHabasit THEN
					// Take results from calibration and save in resultFAT
					resultFAT.CFCaliWithHabasit.ressFrequency := gVibratorInterface[0].status.calibrationResultFrequency;
					resultFAT.CFCaliWithHabasit.maxCurrent := gVibratorInterface[0].status.calibrationResultCurrent;
					resultFAT.CFCaliWithHabasit.currentOK := gVibratorInterface[0].status.calibrationResultCurrentOK;
					resultFAT.CFCaliWithHabasit.frequencyOK := gVibratorInterface[0].status.calibrationResultFrequencyOK;

					resultFAT.CFCaliWithHabasit.strResultForReport := REAL_TO_STRING(resultFAT.CFCaliWithHabasit.maxCurrent);
					resultFAT.LFSpringAdjust.strResultForReport := CONCAT(resultFAT.LFSpringAdjust.strResultForReport,'A');
					resultFAT.CFCaliWithHabasit.strResultForReport := CONCAT(resultFAT.CFCaliWithHabasit.strResultForReport,' / ');
					this.tmpString := REAL_TO_STRING(resultFAT.CFCaliWithHabasit.ressFrequency);
					resultFAT.CFCaliWithHabasit.strResultForReport := CONCAT(resultFAT.CFCaliWithHabasit.strResultForReport,this.tmpString);
					resultFAT.LFSpringAdjust.strResultForReport := CONCAT(resultFAT.LFSpringAdjust.strResultForReport,'Hz');

				END_IF
				this.cfCaliHabasit := FALSE;
			END_IF

			resultFAT.CFCaliWithHabasit.done := resultFAT.CFCaliWithHabasit.currentOK AND resultFAT.CFCaliWithHabasit.frequencyOK;

			IF this.hmi.cmd.arrowNextValue THEN
				this.hmi.cmd.arrowNextValue := FALSE;	// reset.
				state := 190;
			ELSIF this.hmi.cmd.arrowBackValue THEN
				this.hmi.cmd.arrowBackValue := FALSE;
				state := 170;
			END_IF

		190:
			// 12h test

			// 88h test and 12h test
			this.testRunning := this.hmi.testRunning88h XOR this.hmi.testRunning12h;
			gBeltInterface.cmd.runManualTest := gVibratorInterface[0].cmd.runManualTest := gVibratorInterface[1].cmd.runManualTest := this.testRunning;

			IF this.hmi.testRunning88h AND this.hmi.testRunning12h THEN
				// Both can't run at the same time. Disable both if user tries to do this.
				this.hmi.testRunning88h := this.hmi.testRunning12h := FALSE;
			ELSIF this.hmi.testRunning12h THEN

				// Start belt and vibrators
				gBeltInterface.parameter.speedManualTest := 400.0;
				gVibratorInterface[0].parameter.speedPctManualTest := 80.0; // First 12h use 40% rest of the time use 80% (43200s = 12hours)
				gVibratorInterface[1].parameter.speedPctManualTest := 100.0;

				// Calculate time
				this.config.timeElapsed12h := this.config.timeElapsed12h + CYCLE_TIME_seconds;
				this.config.timeLeft12h := 12.0-(this.config.timeElapsed12h/3600);
				this.config.timeLeft12h := getHourMinutsFromDecimal(this.config.timeLeft12h);

				IF this.config.timeLeft12h <= 0.0 THEN
					this.hmi.testRunning12h := this.hmi.testRunning12h := FALSE;
					gConfig.cmd.save := TRUE;
					this.config.timeLeft12h := 0.0;
					resultFAT.longTest12h.done := TRUE;
				END_IF
			END_IF

			// Save to config every 10min
			this.TON_0.IN := this.testRunning;
			this.TON_0.PT := T#10m;
			this.TON_0();

			IF this.TON_0.Q THEN
				this.TON_0.IN := FALSE;
				this.TON_0();

				gConfig.cmd.save := TRUE;
			END_IF

			// If test not running set parameter to 0.
			IF NOT this.testRunning THEN
				gVibratorInterface[0].parameter.speedPctManualTest := 0.0;
				gVibratorInterface[1].parameter.speedPctManualTest := 0.0;
			END_IF

			IF this.hmi.cmd.arrowNextValue THEN
				this.hmi.cmd.arrowNextValue := FALSE;	// reset.
				state := 200;
			ELSIF this.hmi.cmd.arrowBackValue THEN
				this.hmi.cmd.arrowBackValue := FALSE;
				state := 180;
			END_IF

		200:
			// 'Visual inspection of CM marking';

			//	NO SAP LABEL -> resultFAT.visualInspection.markingArr[0]
			//	HAS SAP LABEL -> resultFAT.visualInspection.markingArr[12]

			FOR i:=1 TO 11 DO	// all machine markings must be approved before the step is done.
				IF NOT resultFAT.visualInspection.markingArr[i] THEN
					resultFAT.visualInspection.done := FALSE;
					EXIT;
				ELSIF i=11 THEN
					resultFAT.visualInspection.done := TRUE;

				END_IF
			END_FOR
			IF resultFAT.visualInspection.done THEN
				resultFAT.visualInspection.done :=  resultFAT.visualInspection.markingArr[12] XOR resultFAT.visualInspection.markingArr[0];
			END_IF

			this.hmi.cmd.enableArrowNext := resultFAT.visualInspection.done;

			IF this.hmi.cmd.arrowNextValue THEN
				this.hmi.cmd.arrowNextValue := FALSE;	// reset.
				state := 210;
			ELSIF this.hmi.cmd.arrowBackValue THEN
				this.hmi.cmd.arrowBackValue := FALSE;
				state := 190;
			END_IF

		210:
			// Report and USB transfer (put them together in 1)

			IF this.hmi.status.reportCreationOK AND gMachineInterface.status.configSavedToT50 THEN
				resultFAT.FATdone := TRUE;		// FAT is done!
			END_IF

			generateReportAction;
			usbTransferAction;

			IF this.hmi.cmd.arrowNextValue THEN
				this.hmi.cmd.arrowNextValue := FALSE; // last page cant change state
			ELSIF this.hmi.cmd.arrowBackValue THEN
				this.hmi.cmd.arrowBackValue := FALSE;
				state := 200;
			END_IF

		(*

		10:
			IF gFile.status.ready AND (gConfig.status.saved OR gConfig.status.loaded)  THEN
				this.config.timeLeft88h := 88.0-(this.config.timeElapsed88h/3600);
				this.config.timeLeft88h := getHourMinutsFromDecimal(this.config.timeLeft88h);
				this.config.timeLeft12h := 12.0-(this.config.timeElapsed12h/3600);
				this.config.timeLeft12h := getHourMinutsFromDecimal(this.config.timeLeft12h);

				state := 20;
			END_IF

		20:
			// 88h test and 12h test
			this.testRunning := this.hmi.testRunning88h XOR this.hmi.testRunning12h;
			gBeltInterface.cmd.runManualTest := gVibratorInterface[0].cmd.runManualTest := gVibratorInterface[1].cmd.runManualTest := this.testRunning;

			IF this.hmi.testRunning88h AND this.hmi.testRunning12h THEN
				// Both can't run at the same time. Disable both if user tries to do this.
				this.hmi.testRunning88h := this.hmi.testRunning12h := FALSE;
			ELSIF this.hmi.testRunning88h THEN

				// Start belt and vibrators
				gBeltInterface.parameter.speedManualTest := 400.0;
				gVibratorInterface[0].parameter.speedPctManualTest := SEL(this.config.timeElapsed88h > 43200,40.0,80.0); // First 12h use 40% rest of the time use 80% (43200s = 12hours)
				gVibratorInterface[1].parameter.speedPctManualTest := 100.0;

				// Calculate time
				this.config.timeElapsed88h := this.config.timeElapsed88h + CYCLE_TIME_seconds;
				this.config.timeLeft88h := 88.0-(this.config.timeElapsed88h/3600);
				this.config.timeLeft88h := getHourMinutsFromDecimal(this.config.timeLeft88h);

				IF this.config.timeLeft88h <= 0.0 THEN
					this.hmi.testRunning88h := this.hmi.testRunning12h := FALSE;
					gConfig.cmd.save := TRUE;
					this.config.timeLeft88h := 0.0;
				END_IF
			ELSIF this.hmi.testRunning12h THEN

				// Start belt and vibrators
				gBeltInterface.parameter.speedManualTest := 400.0;
				gVibratorInterface[0].parameter.speedPctManualTest := 80.0; // First 12h use 40% rest of the time use 80% (43200s = 12hours)
				gVibratorInterface[1].parameter.speedPctManualTest := 100.0;

				// Calculate time
				this.config.timeElapsed12h := this.config.timeElapsed12h + CYCLE_TIME_seconds;
				this.config.timeLeft12h := 12.0-(this.config.timeElapsed12h/3600);
				this.config.timeLeft12h := getHourMinutsFromDecimal(this.config.timeLeft12h);

				IF this.config.timeLeft12h <= 0.0 THEN
					this.hmi.testRunning12h := this.hmi.testRunning12h := FALSE;
					gConfig.cmd.save := TRUE;
					this.config.timeLeft12h := 0.0;
				END_IF
			END_IF

			// Save to config every 10min
			this.TON_0.IN := this.testRunning;
			this.TON_0.PT := T#10m;
			this.TON_0();

			IF this.TON_0.Q THEN
				this.TON_0.IN := FALSE;
				this.TON_0();

				gConfig.cmd.save := TRUE;
			END_IF

			// If test not running set parameter to 0.
			IF NOT this.testRunning THEN
				gVibratorInterface[0].parameter.speedPctManualTest := 0.0;
				gVibratorInterface[1].parameter.speedPctManualTest := 0.0;
			END_IF
		*)
	END_CASE

	IF state > 5 THEN
		stateRetain := state;
	END_IF

	IF state > 10 THEN
		// just always allow navigation if we are after state 10 (control of resistance)
		this.hmi.cmd.enableArrowNext := state <> 210; // Disable if last page which is 210 (cant go next on the last page)
	END_IF

	MpRecipeRegPar_Config.MpLink := ADR(mpRecipe);
	MpRecipeRegPar_Config.PVName := ADR(this.configName);
	MpRecipeRegPar_Config.Category := ADR('config');
	MpRecipeRegPar_Config();

	resultsFATfileHandling;

END_PROGRAM

PROGRAM _EXIT
	MpRecipeRegPar_Config.Enable := FALSE;
	MpRecipeRegPar_Config();
	this.MpRecipeRegPar_result.Enable := FALSE;
	this.MpRecipeRegPar_result();
	this.MpReportCore_0.Enable := FALSE;
	this.MpReportCore_0();
END_PROGRAM
```

#### local.typ - Local data types
```iecst
TYPE
	local_typ : 	STRUCT
		configName : STRING[80];
		TON_0 : TON;
		config : config_FAT_typ;
		hmi : local_hmi_typ;
		testRunning : BOOL;
		MpRecipeXml_0 : MpRecipeXml;
		MpRecipeRegPar_result : MpRecipeRegPar;
		ton_chekForChanges : TON;
		resultName : STRING[80];
		resultsFATLoaded : BOOL;
		tmpString : STRING[60];
		oldLREAL : LREAL;
		maxPlusMinusVoltage : REAL := 0.1;
		timeElapsed : UDINT;
		cfCali : BOOL;
		lfCali : BOOL;
		cfCaliHabasit : BOOL;
		hmiUsbPresent : BOOL;
		hmiUsbNotPresent : BOOL;
		fileNameDest : STRING[80];
		folderNameUSB : STRING[80];
		fileNameSrc : STRING[80];
		fileCopy_0 : FileCopy;
		actServerCardIpAddress : STRING[15];
		ftpParamPLC : STRING[80];
		devLinkPLC_0 : DevLink;
		dirPathPLC : STRING[80];
		dirPathUSB : STRING[80];
		dirCopy_0 : DirCopy;
		currentName : STRING[80];
		newName : STRING[80];
		FileRename_0 : FileRename;
		previousState : UINT;
		fileToBeDeleted : STRING[80];
		FileDelete_0 : FileDelete;
		MpReportCore_0 : MpReportCore;
	END_STRUCT;
	local_hmi_typ : 	STRUCT
		testRunning88h : BOOL;
		testRunning12h : BOOL;
		cmd : hmi_cmd_typ;
		status : hmi_status_typ;
		TransferedToUsb : BOOL;
		yearIdx : UINT;
		monthIdx : UINT;
		dayIdx : UINT;
		dateString : STRING[40];
		date : DATE;
	END_STRUCT;
	hmi_cmd_typ : 	STRUCT
		startFAT : BOOL;
		arrowNextValue : BOOL;
		arrowBackValue : BOOL;
		enableMenuNavigation : BOOL;
		enableArrowNext : BOOL;
		smallCfToggleButton : BOOL;
		bigCfToggleButton : BOOL;
		leftDirectionOfRotation : BOOL;
		rightDirectionOfRotation : BOOL;
		crossmarkV2 : USINT;
		crossmarkV1 : USINT;
		startCapconTest2 : BOOL;
		doLevelSensorTest : BOOL;
		setLevelSensorLow : BOOL;
		setLevelSensorMedium : BOOL;
		setLevelSensorHigh : BOOL;
		doPhotoSensorTest : BOOL; (*User wants to start automatic test of the photo sensor.*)
		doPhotoSensorTestNoBelt : BOOL;
		doBfFlapTest : BOOL;
		startLightTowerTest : BOOL;
		doWingTestManuel : BOOL;
		startCalibration : BOOL;
		transferToUsb : BOOL;
		createReports : BOOL;
		transferConfigToFT50 : BOOL;
	END_STRUCT;
	hmi_status_typ : 	STRUCT
		additionalInfo : hmi_status_additionalInfo_typ;
		maxRawSignal : REAL;
		styleToggleInputHigh : BOOL;
		styleToggleInputMedium : BOOL;
		styleToggleInputLow : BOOL;
		photoSensorTestText : USINT;
		isBigMachine : BOOL;
		isSmallMachine : BOOL;
		reportCreationOK : BOOL;
	END_STRUCT;
	hmi_status_additionalInfo_typ : 	STRUCT
		typeNo : UDINT;
		serialNo : UDINT;
		rnoNo : LREAL;
		topSerialNo : UDINT;
		IRTHno : LREAL;
	END_STRUCT;
	config_FAT_typ : 	STRUCT
		timeElapsed88h : REAL;
		timeLeft88h : REAL := 88.0;
		timeElapsed12h : REAL;
		timeLeft12h : REAL := 12.0;
		approveBoltsAreTight : BOOL;
		approveCfHasHabasit : BOOL;
	END_STRUCT;
	permanent_typ : 	STRUCT
		cmState : UINT;
	END_STRUCT;
END_TYPE

(*FAT result structures. Each test point have 1 structs to save results from the test. These are saved on user partition*)

TYPE
	resultFAT_typ : 	STRUCT
		initialGroundMeas : resultFAT_initialGroundMeas_typ;
		machineSetup : resultFAT_machineSetup_typ;
		visualInspection : resultFAT_visualInspection_typ;
		additionalInfo : resultFAT_additionalInfo_typ;
		capconMeasurement : resultFAT_capconMeasurement_typ;
		capconTest : resultFAT_capconTests_typ;
		levelSensorTest : resultFAT_levelSensorTest_typ;
		photoSensorAdjust : resultFAT_photoSensorAdjust_typ;
		photoSensorTest : resultFAT_photoSensorTest_typ;
		bfTestIO : resultFAT_bfTestIO_typ;
		wingTestIO : resultFAT_wingTestIO_typ;
		CFCoilAdjust : resultFAT_CFCoilAdjust_typ;
		CFSpringAdjust : resultFAT_CFSpringAdjust_typ;
		LFCoilAdjust : resultFAT_LFCoildAdjust_typ;
		LFSpringAdjust : resultFAT_LFSpringAdjust_typ;
		longTest88h : resultFAT_88hTest;
		after72hAdjustments : resultFAT_after72hAdjustments;
		CFCaliWithHabasit : resultFAT_CFCaliWithHabasit;
		longTest12h : resultFAT_12hTest;
		resistanceMeas2 : resultFAT_resistanceMeas2_typ;
		internal : internal_typ;
		FATdone : BOOL; (*If all points are done and report has been generated this will be true and FAT is finished.*)
	END_STRUCT;
	resultFAT_initialGroundMeas_typ : 	STRUCT
		done : BOOL;
		measurementValue : REAL;
		firstMeasurementDone : BOOL;
	END_STRUCT;
	resultFAT_machineSetup_typ : 	STRUCT
		done : BOOL;
		cfSize : UINT; (*0 is small, 1 is big*)
		strCfSize : STRING[40];
		strMachineType : STRING[40];
		strMaxSpecsCF : STRING[40]; (*String with current/voltage specs depending of cfSize*)
		strLinearizationAccValuesCF : STRING[40];
		strLinearizationAccValuesLF : STRING[40];
		strIsItALeftMachine : STRING[1]; (*X if yes*)
		strIsItARightMachine : STRING[1]; (*X if yes*)
		machineType : USINT; (*0 is left, 1 is right*)
	END_STRUCT;
	resultFAT_additionalInfo_typ : 	STRUCT
		done : BOOL;
		typeNo : STRING[40];
		serialNo : STRING[40];
		typeNoAndSerialNo : STRING[40];
		vibratorUnitType : STRING[40];
		topUnitType : STRING[40];
		rnaProductNo : STRING[40];
		weightOfCf : STRING[40];
		topSerialNo : STRING[40];
		IRTHno : STRING[40];
	END_STRUCT;
	resultFAT_capconMeasurement_typ : 	STRUCT
		done : BOOL;
		V1 : REAL;
		V2 : REAL;
	END_STRUCT;
	resultFAT_capconTests_typ : 	STRUCT
		done : BOOL;
		signalTest1 : BOOL; (*Test to see if hw signal is comming from capcon to PLC.*)
		signalTest2 : BOOL; (*Test to see if the speed signal is too high. If it is the supply for capcon might be wrong set.*)
	END_STRUCT;
	resultFAT_levelSensorTest_typ : 	STRUCT
		done : BOOL;
		transmitterHighOK : BOOL;
		transmitterMediumOK : BOOL;
		transmitterLowOK : BOOL;
		receiverOK : BOOL;
		operatorApproveHigh : BOOL;
		operatorApproveMedium : BOOL;
		operatorApproveLow : BOOL;
	END_STRUCT;
	resultFAT_photoSensorAdjust_typ : 	STRUCT
		done : BOOL;
	END_STRUCT;
	resultFAT_photoSensorTest_typ : 	STRUCT
		done : BOOL;
		testWithNoBelt : BOOL;
		testWithBelt : BOOL;
	END_STRUCT;
	resultFAT_bfTestIO_typ : 	STRUCT
		done : BOOL;
		approveMainsVoltage : BOOL;
		approveIOsManually : BOOL;
		flapTestDone : BOOL;
	END_STRUCT;
	resultFAT_wingTestIO_typ : 	STRUCT
		done : BOOL;
		correctHartingUsed : BOOL;
		approveFunctionality : BOOL;
		ioTestOK : BOOL;
		upperFlapOK : BOOL;
		middleFlapOK : BOOL;
		bottomFlapOK : BOOL;
		neighbourFlapOK : BOOL;
		cassetteReleaseOK : BOOL;
	END_STRUCT;
	resultFAT_CFCoilAdjust_typ : 	STRUCT
		done : BOOL;
		magneticGap : REAL;
	END_STRUCT;
	resultFAT_CFSpringAdjust_typ : 	STRUCT
		done : BOOL;
		plate08mm : ARRAY[0..2]OF USINT; (*amount of 0.8mm plates on springs (3 springs)*)
		plate09mm : ARRAY[0..2]OF USINT; (*amount of 0.9mm plates on springs (3 springs)*)
		plate15mm : ARRAY[0..2]OF USINT; (*amount of 1.5mm plates on springs (3 springs)*)
		plate20mm : ARRAY[0..2]OF USINT; (*amount of 2.0mm plates on springs (3 springs)*)
		plate25mm : ARRAY[0..2]OF USINT; (*amount of 2.5mm plates on springs (3 springs)*)
		frequency : REAL;
		freqHertz : REAL; (*axis.parameter.velocity/1000*)
		strTargetFrequency : STRING[40]; (*For report to show target frequency interval*)
		ressFrequency : REAL;
		maxCurrent : REAL;
		currentOK : BOOL;
		frequencyOK : BOOL;
	END_STRUCT;
	resultFAT_LFCoildAdjust_typ : 	STRUCT
		done : BOOL;
		magneticGap : REAL;
	END_STRUCT;
	resultFAT_LFSpringAdjust_typ : 	STRUCT
		done : BOOL;
		frequency : REAL;
		freqHertz : REAL; (*axis.parameter.velocity/1000*)
		plate08mm : ARRAY[0..1]OF USINT; (*amount of 0.8mm plates on springs (2 springs)*)
		plate09mm : ARRAY[0..1]OF USINT; (*amount of 0.8mm plates on springs (2 springs)*)
		plate15mm : ARRAY[0..1]OF USINT; (*amount of 0.8mm plates on springs (2 springs)*)
		plate20mm : ARRAY[0..1]OF USINT; (*amount of 0.8mm plates on springs (2 springs)*)
		plate25mm : ARRAY[0..1]OF USINT; (*amount of 0.8mm plates on springs (2 springs)*)
		ressFrequency : REAL;
		maxCurrent : REAL;
		currentOK : BOOL;
		frequencyOK : BOOL;
		strResultForReport : STRING[80];
	END_STRUCT;
	resultFAT_88hTest : 	STRUCT
		done : BOOL;
	END_STRUCT;
	resultFAT_after72hAdjustments : 	STRUCT
		done : BOOL;
		approvePacemakerMarking : BOOL;
		approveCoverMounting : BOOL;
		approveRNAmarking : BOOL;
		approveHabasitMounting : BOOL;
	END_STRUCT;
	resultFAT_CFCaliWithHabasit : 	STRUCT
		done : BOOL;
		ressFrequency : REAL;
		maxCurrent : REAL;
		currentOK : BOOL;
		frequencyOK : BOOL;
		strResultForReport : STRING[80];
	END_STRUCT;
	resultFAT_12hTest : 	STRUCT
		done : BOOL;
	END_STRUCT;
	resultFAT_resistanceMeas2_typ : 	STRUCT
		done : BOOL;
		measurementArr : ARRAY[0..8]OF REAL;
		measurementOK : {REDUND_UNREPLICABLE} ARRAY[0..8]OF BOOL;
	END_STRUCT;
	resultFAT_visualInspection_typ : 	STRUCT
		done : BOOL;
		markingArr : ARRAY[0..12]OF BOOL; (*11 marks to check*)
	END_STRUCT;
	internal_typ : 	STRUCT  (*Internal variables that are saved in a file (used because retain memory sometimes get flushed doing a power fail)*)
		emSubstate : UINT;
		testProgramVersion : STRING[80];
	END_STRUCT;
END_TYPE
```

#### local.var - Local variables
```iecst
VAR CONSTANT
	CYCLE_TIME_seconds : REAL := 0.04;
END_VAR
VAR
	MpRecipeRegPar_Config : MpRecipeRegPar;
	this : local_typ;
	state : UINT;
END_VAR
VAR RETAIN
	stateRetain : UINT;
END_VAR
VAR
	resultFATOld : resultFAT_typ;
	resultFAT : resultFAT_typ; (*Will store the results doing FAT.*)
	i : USINT;
	stateRecipe : UINT;
	levelTestState : USINT;
	nodeIdList : ARRAY[0..4] OF UDINT;
	UsbNodeListGet_0 : UsbNodeListGet;
	usbState : UINT;
	buffer : usbNode_typ;
	UsbNodeGet_0 : UsbNodeGet;
	paramString : STRING[80];
	DevLink_0 : DevLink;
	dirCreate_0 : DirCreate;
	reportState : UINT;
END_VAR
```

#### LocalFunctions.fun
```iecst
{REDUND_ERROR} FUNCTION getHourMinutsFromDecimal : REAL (*TODO: Add your comment here*) (*$GROUP=User,$CAT=User,$GROUPICON=User.png,$CATICON=User.png*)
	VAR_INPUT
		decimalTime : REAL;
	END_VAR
	VAR
		hours : INT;
		minutes : INT;
	END_VAR
END_FUNCTION
```

#### getHourMinutsFromDecimal.st
```iecst
(* TODO: Add your comment here *)
FUNCTION getHourMinutsFromDecimal

	hours := TRUNC(decimalTime);
	minutes := TRUNC((decimalTime - hours) * 60);

	getHourMinutsFromDecimal := INT_TO_REAL(hours)+INT_TO_REAL(minutes)/100;

END_FUNCTION
```

#### resultsFATfileHandling.st
```iecst
ACTION resultsFATfileHandling:

	CASE stateRecipe OF

		0:
		//	cm.description := 'wait for file devices to be ready';

			IF gFile.status.ready AND gConfig.status.loaded THEN
				this.MpRecipeRegPar_result.Enable := TRUE;
				stateRecipe := 10;
			END_IF

		10:
	//		cm.description := 'wait for MpRecipeXml to be active';

			this.MpRecipeXml_0.Enable := TRUE;
			IF this.MpRecipeXml_0.Active THEN
				stateRecipe := 100;
			ELSIF this.MpRecipeXml_0.Error THEN
				stateRecipe := 9999;
			END_IF

		100:
		//	cm.description := 'wait for load or save command';

			IF this.MpRecipeXml_0.Load THEN
				stateRecipe := 200;
			ELSIF this.MpRecipeXml_0.Save THEN
				stateRecipe := 300;
			END_IF

		200:
		//	cm.description := 'wait for loading file';

			IF this.MpRecipeXml_0.CommandDone THEN
				// reset the load cmd
				this.MpRecipeXml_0.Load := FALSE;
				resultFATOld := resultFAT; // After load update old (no reason to save immediatly after)
				this.resultsFATLoaded := TRUE;
				stateRecipe := 100;
			ELSIF this.MpRecipeXml_0.Error THEN
				this.MpRecipeXml_0.Load := FALSE;
				CASE this.MpRecipeXml_0.StatusID OF

					-1064140798,-1064140791: // mpRECIPE_ERR_LOAD_DATA
						this.MpRecipeXml_0.ErrorReset := TRUE;
						stateRecipe := 210;

					ELSE
						stateRecipe := 9999;
				END_CASE
			END_IF

		210:
		//	cm.description := 'wait for NOT MpRecipeXml_0.Error';

			IF NOT this.MpRecipeXml_0.Error THEN
				this.MpRecipeXml_0.ErrorReset := FALSE;
				this.MpRecipeXml_0.Save := TRUE;
				stateRecipe := 300;
			END_IF

		300:
		//	cm.description := 'wait for saving file';

			IF this.MpRecipeXml_0.CommandDone THEN
				// reset the save cmd
				this.MpRecipeXml_0.Save := FALSE;
				this.resultsFATLoaded := TRUE; // If saved also say that we have loaded (first download when file is not there)
				stateRecipe := 100;
			ELSIF this.MpRecipeXml_0.Error THEN
				this.MpRecipeXml_0.Save := FALSE;
				stateRecipe := 9999;
			END_IF

		9999:
		//	cm.description := 'wait for error reset';

			IF NOT this.MpRecipeXml_0.Error THEN
				stateRecipe := 10;
			END_IF

	END_CASE

	this.MpRecipeXml_0.MpLink := ADR(mpResult);
	this.MpRecipeXml_0.DeviceName := ADR('RESULT');
	this.MpRecipeXml_0.FileName := ADR('result.xml');
	this.MpRecipeXml_0.Category := ADR('result');
	this.MpRecipeXml_0();

	// Check if resultsFAT has changed with a TON
	this.ton_chekForChanges(IN:=NOT this.MpRecipeXml_0.Save AND NOT this.MpRecipeXml_0.Load);

	IF this.ton_chekForChanges.Q THEN
		this.ton_chekForChanges(IN:=FALSE);

		IF brsmemcmp(ADR(resultFAT),ADR(resultFATOld),SIZEOF(resultFATOld)) <> 0 THEN
			this.MpRecipeXml_0.Save := TRUE;
		END_IF
		resultFATOld := resultFAT;

	END_IF
	this.MpRecipeRegPar_result(MpLink := ADR(mpResult), PVName := ADR(this.resultName), Category := ADR('result'));

END_ACTION
```

#### usbTransferAction.st
```iecst
ACTION usbTransferAction:

		//-----------------------------------------------------
			//----------------- USB Handling ----------------------
			//-----------------------------------------------------
	UsbNodeListGet_0.enable 		:= TRUE;
	UsbNodeListGet_0.pBuffer 		:= ADR(nodeIdList);
	UsbNodeListGet_0.bufferSize 	:= SIZEOF(nodeIdList);
	UsbNodeListGet_0();

	IF UsbNodeListGet_0.status <> ERR_FUB_BUSY THEN

		IF UsbNodeListGet_0.status = ERR_OK THEN
			this.hmiUsbPresent := TRUE;
			this.hmiUsbNotPresent := FALSE;
		ELSE
			this.hmiUsbPresent := FALSE;
			this.hmiUsbNotPresent := TRUE;
		END_IF

	END_IF

	CASE usbState OF

		0:
			IF this.hmi.cmd.transferToUsb THEN
				this.hmi.cmd.transferToUsb := FALSE;
				this.hmi.TransferedToUsb := FALSE;
				usbState := 10;
			END_IF

		10:	// wait for node list ready
			IF UsbNodeListGet_0.status = ERR_OK THEN
				UsbNodeGet_0(enable 	:= FALSE);
				UsbNodeGet_0.enable 	:= TRUE;
				UsbNodeGet_0.nodeId 	:= nodeIdList[0];
				UsbNodeGet_0.pBuffer 	:= ADR(buffer);
				UsbNodeGet_0.bufferSize := SIZEOF(buffer);
				usbState := 20;
			END_IF

		20:	// get usb info
			UsbNodeGet_0();
			IF UsbNodeGet_0.status = ERR_OK THEN
				DevLink_0(enable := FALSE);
				paramString := '/DEVICE=';
				brdkStrCat(ADR(paramString),ADR(buffer.ifName));
				DevLink_0.pDevice 	:= ADR('USB');
				DevLink_0.pParam 	:= ADR(paramString);
				DevLink_0.enable 	:= TRUE;
				usbState		:= 30;
			END_IF

		30:	// get dev link
			DevLink_0();
			IF DevLink_0.status = ERR_OK OR DevLink_0.status = fiERR_DEVICE_ALREADY_EXIST THEN
				DevLink_0(enable := FALSE);

				IF resultFAT.additionalInfo.typeNoAndSerialNo='' THEN
					this.fileNameDest := 'DataCM20';
				ELSE
					this.fileNameDest := resultFAT.additionalInfo.typeNoAndSerialNo;
					this.tmpString := 'DataCM20';
					brdkStrCat(ADR(this.fileNameDest),ADR(this.tmpString));
				END_IF

				usbState := 40;
			END_IF

		40: // dir create
			//	 'Create a folder on USB before we dirCopy';

			dirCreate_0.enable := TRUE;
			dirCreate_0.pDevice := ADR('USB');
			dirCreate_0.pName := ADR(this.fileNameDest);
			dirCreate_0();

			IF dirCreate_0.status = ERR_OK OR dirCreate_0.status = fiERR_DIR_ALREADY_EXIST  THEN
				dirCreate_0(enable := FALSE);
				this.folderNameUSB := this.fileNameDest;
				this.fileNameSrc := 'config.xml';
				IF resultFAT.additionalInfo.typeNoAndSerialNo='' THEN
					this.fileNameDest := 'DataCM20\config.xml';
				ELSE
					this.tmpString := '\';
					brdkStrCat(ADR(this.fileNameDest),ADR(this.tmpString));
					this.tmpString := resultFAT.additionalInfo.typeNoAndSerialNo;
					brdkStrCat(ADR(this.fileNameDest),ADR(this.tmpString));
					this.tmpString := 'config.xml';
					brdkStrCat(ADR(this.fileNameDest),ADR(this.tmpString));
				END_IF
				usbState := 50;
			ELSIF dirCreate_0.status <> ERR_FUB_BUSY THEN
				dirCreate_0(enable := FALSE);
				usbState := 9999;
			END_IF

		50: // copy config file
			this.fileCopy_0.enable := TRUE;
			this.fileCopy_0.pSrcDev := ADR('CONFIG');
			this.fileCopy_0.pSrc := ADR(this.fileNameSrc);
			this.fileCopy_0.pDestDev := ADR('USB');
			this.fileCopy_0.pDest := ADR(this.fileNameDest);
			this.fileCopy_0.option := fiOVERWRITE;
			this.fileCopy_0();

			IF this.fileCopy_0.status = ERR_OK THEN
				this.fileCopy_0(enable := FALSE);
				// Create ftp param for PLC devlink creation.
				this.actServerCardIpAddress := '192.168.2.11';
				this.ftpParamPLC := '/SIP=';
				brdkStrCat(ADR(this.ftpParamPLC),ADR(this.actServerCardIpAddress));
				this.tmpString := ' /PROTOCOL=ftp /USER=superuser /PASSWORD=superuser';
				brdkStrCat(ADR(this.ftpParamPLC),ADR(this.tmpString));
				usbState := 55;
			ELSIF this.fileCopy_0.status <> ERR_FUB_BUSY THEN
				usbState := 9999;
			END_IF

		55: // create plc dev link
			this.devLinkPLC_0.enable := TRUE;
			this.devLinkPLC_0.pDevice := ADR('PLC');
			this.devLinkPLC_0.pParam := ADR(this.ftpParamPLC);
			this.devLinkPLC_0();
			IF this.devLinkPLC_0.status=0 OR this.devLinkPLC_0.status=fiERR_DEVICE_ALREADY_EXIST THEN	// devLink created successfully or it's already created.
				this.devLinkPLC_0(enable := FALSE);
				this.dirPathPLC := 'F:\data';
				IF resultFAT.additionalInfo.typeNoAndSerialNo='' THEN
					this.dirPathUSB := 'DataCM20\data';
				ELSE
					this.dirPathUSB := this.folderNameUSB;
					this.tmpString := '\';
					brdkStrCat(ADR(this.dirPathUSB),ADR(this.tmpString));
					this.tmpString := resultFAT.additionalInfo.typeNoAndSerialNo;
					brdkStrCat(ADR(this.dirPathUSB),ADR(this.tmpString));
					this.tmpString := 'data';
					brdkStrCat(ADR(this.dirPathUSB),ADR(this.tmpString));
				END_IF
				usbState := 60;
			ELSIF this.devLinkPLC_0.status <> ERR_FUB_BUSY THEN
				this.devLinkPLC_0(enable := FALSE);
				usbState := 9999;
			END_IF

		60:
			// 'Copy data DIR to usb';

			this.dirCopy_0.enable := TRUE;
			this.dirCopy_0.pSrcDev := ADR('PLC');
			this.dirCopy_0.pSrcDir := ADR(this.dirPathPLC);
			this.dirCopy_0.pDestDev := ADR('USB');
			this.dirCopy_0.pDestDir := ADR(this.dirPathUSB);
			this.dirCopy_0.option := fiOVERWRITE;
			this.dirCopy_0();

			IF this.dirCopy_0.status = 0 THEN
				this.dirCopy_0(enable := FALSE);
				this.dirPathPLC := 'F:\report';
				IF resultFAT.additionalInfo.typeNoAndSerialNo='' THEN
					this.dirPathUSB := 'DataCM20\report';
				ELSE
					this.dirPathUSB := this.folderNameUSB;
					this.tmpString := '\';
					brdkStrCat(ADR(this.dirPathUSB),ADR(this.tmpString));
					this.tmpString := resultFAT.additionalInfo.typeNoAndSerialNo;
					brdkStrCat(ADR(this.dirPathUSB),ADR(this.tmpString));
					this.tmpString := 'reports';
					brdkStrCat(ADR(this.dirPathUSB),ADR(this.tmpString));
				END_IF
				usbState := 70;
			ELSIF this.dirCopy_0.status <> ERR_FUB_BUSY THEN
				this.dirCopy_0(enable := FALSE);
				usbState := 9999;
			END_IF

		70:
			// 'Copy report DIR to usb';

			this.dirCopy_0.enable := TRUE;
			this.dirCopy_0.pSrcDev := ADR('PLC');
			this.dirCopy_0.pSrcDir := ADR(this.dirPathPLC);
			this.dirCopy_0.pDestDev := ADR('USB');
			this.dirCopy_0.pDestDir := ADR(this.dirPathUSB);
			this.dirCopy_0.option := fiOVERWRITE;
			this.dirCopy_0();

			IF this.dirCopy_0.status = 0 THEN
				this.dirCopy_0(enable := FALSE);
				IF resultFAT.additionalInfo.typeNoAndSerialNo = '' THEN
					this.hmi.TransferedToUsb := TRUE;
					this.hmi.cmd.transferToUsb := FALSE;
					usbState := 0;
				ELSE
					// create names for rename
					this.currentName := this.dirPathUSB; //report path on USB
					this.tmpString := '\CM20Protocol.pdf';
					brdkStrCat(ADR(this.currentName),ADR(this.tmpString));
					// New name
					this.newName := this.dirPathUSB;
					this.tmpString := '\';
					brdkStrCat(ADR(this.newName),ADR(this.tmpString));
					this.tmpString := resultFAT.additionalInfo.typeNoAndSerialNo;
					brdkStrCat(ADR(this.newName),ADR(this.tmpString));
					this.tmpString := 'CM20Protocol.pdf';
					brdkStrCat(ADR(this.newName),ADR(this.tmpString));

					usbState := 72;
				END_IF
			ELSIF this.dirCopy_0.status <> ERR_FUB_BUSY THEN
				this.dirCopy_0(enable := FALSE);
				usbState := 9999;
			END_IF

		72:
			// 'Rename protocol report';

			this.FileRename_0.enable := TRUE;
			this.FileRename_0.pDevice := ADR('USB');
			this.FileRename_0.pName := ADR(this.currentName);
			this.FileRename_0.pNewName := ADR(this.newName);
			this.FileRename_0();

			IF this.FileRename_0.status = 0 THEN
				this.FileRename_0(enable:=FALSE);
				// create names for rename
				this.currentName := this.dirPathUSB; //report path on USB
				this.tmpString := '\CM20Checklist.pdf';
				brdkStrCat(ADR(this.currentName),ADR(this.tmpString));
				// New name
				this.newName := this.dirPathUSB;
				this.tmpString := '\';
				brdkStrCat(ADR(this.newName),ADR(this.tmpString));
				this.tmpString := resultFAT.additionalInfo.typeNoAndSerialNo;
				brdkStrCat(ADR(this.newName),ADR(this.tmpString));
				this.tmpString := 'CM20Checklist.pdf';
				brdkStrCat(ADR(this.newName),ADR(this.tmpString));

				usbState := 74;

			ELSIF this.FileRename_0.status=fiERR_EXIST THEN
				this.FileRename_0(enable:=FALSE);
				this.previousState := usbState;
				this.fileToBeDeleted := this.newName;

				usbState := 222;
			ELSIF this.FileRename_0.status <> ERR_FUB_BUSY THEN
				this.FileRename_0(enable:=FALSE);
				usbState := 9999;
			END_IF

		74:
			// 'Rename checklist report';

			this.FileRename_0.enable := TRUE;
			this.FileRename_0.pDevice := ADR('USB');
			this.FileRename_0.pName := ADR(this.currentName);
			this.FileRename_0.pNewName := ADR(this.newName);
			this.FileRename_0();

			IF this.FileRename_0.status = 0 THEN
				this.FileRename_0(enable:=FALSE);
				// create names for rename
				this.currentName := this.dirPathUSB; //report path on USB
				this.tmpString := '\CM20hwReport.pdf';
				brdkStrCat(ADR(this.currentName),ADR(this.tmpString));
				// New name
				this.newName := this.dirPathUSB;
				this.tmpString := '\';
				brdkStrCat(ADR(this.newName),ADR(this.tmpString));
				this.tmpString := resultFAT.additionalInfo.typeNoAndSerialNo;
				brdkStrCat(ADR(this.newName),ADR(this.tmpString));
				this.tmpString := 'CM20hwReport.pdf';
				brdkStrCat(ADR(this.newName),ADR(this.tmpString));

				usbState := 76;
			ELSIF this.FileRename_0.status=fiERR_EXIST THEN
				this.FileRename_0(enable:=FALSE);
				this.previousState := usbState;
				this.fileToBeDeleted := this.newName;

				usbState := 222;
			ELSIF this.FileRename_0.status <> ERR_FUB_BUSY THEN
				this.FileRename_0(enable:=FALSE);
				usbState := 9999;
			END_IF

		76:
			// 'Rename hw report';

			this.hmi.TransferedToUsb := TRUE;
			this.hmi.cmd.transferToUsb := FALSE;

			usbState := 0;

		222:
			//'Delete file and return to previous state';

			this.FileDelete_0.enable := TRUE;
			this.FileDelete_0.pDevice := ADR('USB');
			this.FileDelete_0.pName := ADR(this.fileToBeDeleted);
			this.FileDelete_0();

			IF this.FileDelete_0.status=0 THEN
				this.FileDelete_0(enable:=FALSE);
				usbState := this.previousState;
			ELSIF this.FileDelete_0.status <> ERR_FUB_BUSY THEN
				this.FileDelete_0(enable:=FALSE);
				usbState := 9999;
			END_IF

		9999:
			UsbNodeListGet_0(enable := FALSE);
			UsbNodeGet_0(enable := FALSE);
			this.FileRename_0(enable:=FALSE);
			this.dirCopy_0(enable := FALSE);
			this.devLinkPLC_0(enable := FALSE);
			this.fileCopy_0(enable := FALSE);

			usbState := 0;

	END_CASE

END_ACTION
```

#### generateReportAction.st
```iecst
ACTION generateReportAction:

	CASE reportState OF

		0:
		//	'Wait for user to input cmd';
			this.MpReportCore_0.Enable := FALSE;

			IF this.hmi.cmd.createReports THEN
				this.hmi.cmd.createReports := FALSE;
				this.hmi.status.reportCreationOK := FALSE;
				resultFAT.FATdone := FALSE;

				gMachineInterface.cmd.saveConfigToT50 := TRUE;
				//Generate data from user input:
				this.hmi.dateString := '';
				brdkStrCat(ADR(this.hmi.dateString),ADR('D#'));
				this.hmi.yearIdx := 2020+this.hmi.yearIdx;	// 0 means 2020
				this.tmpString := UINT_TO_STRING(this.hmi.yearIdx);
				brdkStrCat(ADR(this.hmi.dateString),ADR(this.tmpString));
				brdkStrCat(ADR(this.hmi.dateString),ADR('-'));

				this.hmi.monthIdx := 1+this.hmi.monthIdx;	//0 means 1 (january)
				IF this.hmi.monthIdx < 10 THEN
					this.tmpString := '0';
					brdkStrCat(ADR(this.hmi.dateString),ADR(this.tmpString));
				END_IF
				this.tmpString := UINT_TO_STRING(this.hmi.monthIdx);
				brdkStrCat(ADR(this.hmi.dateString),ADR(this.tmpString));
				brdkStrCat(ADR(this.hmi.dateString),ADR('-'));

				this.hmi.dayIdx := 1+this.hmi.dayIdx; 		// 0 means day 1
				IF this.hmi.dayIdx < 10 THEN
					this.tmpString := '0';
					brdkStrCat(ADR(this.hmi.dateString),ADR(this.tmpString));
				END_IF
				this.tmpString := UINT_TO_STRING(this.hmi.dayIdx);
				brdkStrCat(ADR(this.hmi.dateString),ADR(this.tmpString));
				this.hmi.date := STRING_TO_DATE(this.hmi.dateString);

				// gReport cmd will we reset in hwReadout task
				this.MpReportCore_0.Enable := TRUE;

				this.ftpParamPLC := '/SIP=192.168.2.11 /PROTOCOL=ftp /USER=superuser /PASSWORD=superuser';
				reportState := 10;
			END_IF

		10:
			// 'Create devlink to PLC';

			this.devLinkPLC_0.enable := TRUE;
			this.devLinkPLC_0.pDevice := ADR('PLC');
			this.devLinkPLC_0.pParam := ADR(this.ftpParamPLC);
			this.devLinkPLC_0();

			IF this.devLinkPLC_0.status=0 OR this.devLinkPLC_0.status=fiERR_DEVICE_ALREADY_EXIST THEN	// devLink created successfully or it's already created.
				this.devLinkPLC_0.enable := FALSE;
				this.devLinkPLC_0();
				// Go to state where we move images from PLC to IMAGES file device.
				this.fileNameSrc := 'C:\ADDONS\DATA\IAT_Data\wwwRoot\BRVisu\Media\Images\leftMachine.jpg';
				this.fileNameDest := 'leftMachine.jpg';
				reportState := 20;
			END_IF

		20:
			this.fileCopy_0.enable := TRUE;
			this.fileCopy_0.pSrcDev := ADR('PLC');
			this.fileCopy_0.pSrc := ADR(this.fileNameSrc);
			this.fileCopy_0.pDestDev := ADR('IMAGES');
			this.fileCopy_0.pDest := ADR(this.fileNameDest);
			this.fileCopy_0.option := fiOVERWRITE;
			this.fileCopy_0();

			IF this.fileCopy_0.status = ERR_OK THEN
				this.fileCopy_0(enable := FALSE);
				this.fileNameSrc := 'C:\ADDONS\DATA\IAT_Data\wwwRoot\BRVisu\Media\Images\rightMachine.jpg';
				this.fileNameDest := 'rightMachine.jpg';
				reportState := 30;
			END_IF

		30:
			this.fileCopy_0.enable := TRUE;
			this.fileCopy_0.pSrcDev := ADR('PLC');
			this.fileCopy_0.pSrc := ADR(this.fileNameSrc);
			this.fileCopy_0.pDestDev := ADR('IMAGES');
			this.fileCopy_0.pDest := ADR(this.fileNameDest);
			this.fileCopy_0.option := fiOVERWRITE;
			this.fileCopy_0();

			IF this.fileCopy_0.status = ERR_OK THEN
				this.fileCopy_0(enable := FALSE);
				reportState := 40; // Done moving pics
			END_IF

		40:
			IF this.MpReportCore_0.Active THEN
				reportState := 50;
			END_IF

		50:
			this.MpReportCore_0.Name := ADR('CM20Protocol');
			this.MpReportCore_0.Generate := TRUE;

			IF this.MpReportCore_0.CommandDone THEN
				this.MpReportCore_0.Generate := FALSE;
				reportState := 60;
			ELSIF this.MpReportCore_0.Error THEN
				this.MpReportCore_0.Generate := FALSE;
				reportState := 9999;
			END_IF

		60:
			// 'Generate checklist';

			this.MpReportCore_0.Name := ADR('CM20Checklist');
			this.MpReportCore_0.Generate := TRUE;

			IF this.MpReportCore_0.CommandDone THEN
				this.MpReportCore_0.Generate := FALSE;
				this.hmi.status.reportCreationOK := TRUE;
				// Reports generated. Trigger a factory reset to be sure parameters are optimal.
				gConfig.status.factoryReset[0] := gConfig.status.factoryReset[1] := gConfig.status.factoryReset[2] := gConfig.status.factoryReset[3] := gConfig.status.factoryReset[4] := TRUE;
				reportState := 0;
			ELSIF this.MpReportCore_0.Error THEN
				this.MpReportCore_0.Generate := FALSE;
				reportState := 9999;
			END_IF

		9999:
			// 'Error';
			this.hmi.status.reportCreationOK := FALSE;

			IF NOT this.MpReportCore_0.Error THEN
				reportState := 0;
			END_IF

	END_CASE

	this.MpReportCore_0.MpLink := ADR(mpReport);
	this.MpReportCore_0.Language := ADR('en');
	this.MpReportCore_0.DeviceName := ADR('REPORT');
	this.MpReportCore_0();

END_ACTION
```

### Program Logical/simulation/simulation (IEC)

#### main.st - Init, cyclic, exit code
```iecst
PROGRAM _INIT

//	gSimulation.status.simulateAllButWing := TRUE; // REMOVE BEFORE PRODUCTION

END_PROGRAM

PROGRAM _CYCLIC

	IF gMainInterface.status.simulation THEN
		capcon.activated := TRUE;
		feeder.activated := TRUE;
		belt.activated := TRUE;
		wing.activated := TRUE;
		cassette.activated := TRUE;
		vision.activated := TRUE;
	ELSIF gSimulation.status.simulateAllButWing THEN
		capcon.activated := TRUE;
		feeder.activated := FALSE;
		belt.activated := TRUE;
		wing.activated := FALSE;
		cassette.activated := FALSE;
		vision.activated := FALSE;
	ELSE
		capcon.activated := FALSE;
		feeder.activated := FALSE;
		belt.activated := FALSE;
		wing.activated := FALSE;
		cassette.activated := FALSE;
		vision.activated := FALSE;
	END_IF

	//vibrator; // remove warning

	cassette.activated := gWingInterface.status.simCassette;

	//simulation of feeder
	simFeeder;

	//simulation of vibrator
	//simVibrator;

	//simulation of belt
	simBelt;

	//simulation of capcon
	simCapcon;

	//simulation of wing unit
	//simWing;

	//simulation of cassette
	simCassette;

END_PROGRAM

PROGRAM _EXIT
	FOR i:=0 TO MAX_INPUT_CASSETTE DO
		cassette.hw.in[i](enable := FALSE);
	END_FOR
	FOR i:=0 TO MAX_OUTPUT_CASSETTE DO
		cassette.hw.out[i](enable := FALSE);
	END_FOR

END_PROGRAM
```

#### types.typ - Local data types
```iecst
TYPE
	local_feeder_typ : 	STRUCT
		activated : BOOL;
		var : local_feeder_var_typ;
		hw : local_feeder_hw_typ;
	END_STRUCT;
	local_feeder_var_typ : 	STRUCT
		TOF_levelSensorOn : TOF;
		TON_levelSensorOff : TON;
		TON_0 : TON;
		flapSpeed : REAL;
		stateFlap : USINT;
	END_STRUCT;
	local_feeder_hw_typ : 	STRUCT
		in : ARRAY[0..MAX_INPUT_FEEDER]OF brdkSimInput;
		out : ARRAY[0..MAX_OUTPUT_FEEDER]OF brdkSimOutput;
	END_STRUCT;
	local_vibrator_typ : 	STRUCT
		activated : BOOL;
		var : local_vibrator_var_typ;
		hw : local_vibrator_hw_typ;
	END_STRUCT;
	local_vibrator_var_typ : 	STRUCT
		TON_sensor : TON;
		flapSpeed : REAL;
		state : USINT;
	END_STRUCT;
	local_vibrator_hw_typ : 	STRUCT
		in : ARRAY[0..MAX_INPUT_VIBRATOR]OF brdkSimInput;
		out : ARRAY[0..MAX_OUTPUT_VIBRATOR]OF brdkSimOutput;
	END_STRUCT;
	local_belt_typ : 	STRUCT
		activated : BOOL;
		usePWMforSim : BOOL;
		var : local_belt_var_typ;
		hw : local_belt_hw_typ;
	END_STRUCT;
	local_belt_var_typ : 	STRUCT
		convPosition : REAL;
		TON_sensor : TON;
		convSpeed : REAL;
		state : UINT;
		brickLength : REAL := 20;
		brickStart : REAL;
		gapLength : REAL := 50;
		brickGap : REAL;
		gapLengthVarMax : UDINT;
		gapLengthVarMin : UDINT;
		gapVariancePrc : REAL := 0.3;
		gapStart : REAL;
		brickEnd : REAL;
		bricksAtEdgeIdx : UINT;
		bricksAtEdge : ARRAY[0..299]OF REAL;
		percentToSpeed : REAL := 1;
	END_STRUCT;
	local_belt_hw_typ : 	STRUCT
		in : ARRAY[0..MAX_INPUT_BELT]OF brdkSimInput;
		out : ARRAY[0..MAX_OUTPUT_BELT]OF brdkSimOutput;
	END_STRUCT;
	local_capcon_typ : 	STRUCT
		activated : BOOL;
		var : local_capcon_var_typ;
		hw : local_capcon_hw_typ;
	END_STRUCT;
	local_capcon_var_typ : 	STRUCT
		i : UINT;
		j : UINT;
		oldSensor : UDINT;
		state : USINT;
		line : STRING[1000000];
		data : ARRAY[0..99]OF local_capcon_var_data_typ;
		setInputValue : INT;
		setInputValueR : REAL;
		beltPosition : REAL;
		signalIdx : UINT;
		signals : ARRAY[0..299]OF INT;
		x : REAL;
		currSignal : REAL;
		signalHeight : REAL := 1000;
		errorRate : REAL := 0.0;
		rejects : ARRAY[0..299]OF BOOL;
	END_STRUCT;
	local_capcon_var_data_typ : 	STRUCT
		brick : ARRAY[0..499]OF INT;
	END_STRUCT;
	local_capcon_hw_typ : 	STRUCT
		in : ARRAY[0..MAX_INPUT_CAPCON]OF brdkSimInput;
		out : ARRAY[0..MAX_OUTPUT_CAPCON]OF brdkSimOutput;
	END_STRUCT;
	local_wing_typ : 	STRUCT
		activated : BOOL;
		var : local_wing_var_typ;
		hw : local_wing_hw_typ;
	END_STRUCT;
	local_wing_var_typ : 	STRUCT
		oldVal : ARRAY[0..MAX_WINGS]OF UDINT;
		TON_delay : ARRAY[0..MAX_WINGS]OF TON;
		TOF_changeOver : ARRAY[0..MAX_WINGS]OF TOF;
	END_STRUCT;
	local_wing_hw_typ : 	STRUCT
		in : ARRAY[0..MAX_INPUT_WING]OF brdkSimInput;
		out : ARRAY[0..MAX_OUTPUT_WING]OF brdkSimOutput;
	END_STRUCT;
	local_cassette_typ : 	STRUCT
		activated : BOOL;
		var : local_cassette_var_typ;
		hw : local_cassette_hw_typ;
	END_STRUCT;
	local_cassette_var_typ : 	STRUCT
		cassetteInPlace : BOOL;
		tonDelay : TON := (PT:=T#0ms);
		state : USINT;
		toReadyTime : TIME := T#560ms;
		fromReadyTime : TIME := T#67ms;
		fromQueueTime : TIME := T#300ms;
		cassetteQueueTime : TIME := T#1s;
		tofDelay : TOF;
	END_STRUCT;
	local_cassette_hw_typ : 	STRUCT
		in : ARRAY[0..MAX_INPUT_CASSETTE]OF brdkSimInput;
		out : ARRAY[0..MAX_OUTPUT_CASSETTE]OF brdkSimOutput;
	END_STRUCT;
	local_external_typ : 	STRUCT
		activated : BOOL;
		var : local_external_var_typ;
		hw : local_external_hw_typ;
	END_STRUCT;
	local_external_var_typ : 	STRUCT
		dummy : USINT;
	END_STRUCT;
	local_external_hw_typ : 	STRUCT
		in : ARRAY[0..MAX_INPUT_EXTERNAL]OF brdkSimInput;
		out : ARRAY[0..MAX_OUTPUT_EXTERNAL]OF brdkSimOutput;
	END_STRUCT;
	local_vision_typ : 	STRUCT
		activated : BOOL;
		var : local_vision_var_typ;
		hw : local_vision_hw_typ;
	END_STRUCT;
	local_vision_var_typ : 	STRUCT
		New_Member : USINT;
	END_STRUCT;
	local_vision_hw_typ : 	STRUCT
		in : ARRAY[0..MAX_INPUT_VISION]OF brdkSimInput;
		out : ARRAY[0..MAX_OUTPUT_VISION]OF brdkSimOutput;
	END_STRUCT;
END_TYPE
```

#### variables.var - Local variables
```iecst
VAR
	i : USINT;
	feeder : local_feeder_typ;
	belt : local_belt_typ;
	capcon : local_capcon_typ;
	wing : local_wing_typ;
	vision : local_vision_typ; (*external : local_external_typ;*)
	cassette : local_cassette_typ; (*external : local_external_typ;*)
END_VAR
VAR CONSTANT
	MAX_INPUT_FEEDER : USINT := 4;
	MAX_INPUT_VIBRATOR : USINT := 0;
	MAX_INPUT_VISION : USINT := 0;
	MAX_INPUT_BELT : USINT := 0;
	MAX_INPUT_CAPCON : USINT := 0;
	MAX_WINGS : USINT := 3;
	MAX_INPUT_WING : USINT := 5;
	MAX_INPUT_CASSETTE : USINT := 2;
	MAX_INPUT_EXTERNAL : USINT := 0;
	MAX_OUTPUT_FEEDER : USINT := 2;
	MAX_OUTPUT_VIBRATOR : USINT := 0;
	MAX_OUTPUT_VISION : USINT := 0;
	MAX_OUTPUT_BELT : USINT := 0;
	MAX_OUTPUT_CAPCON : USINT := 0;
	MAX_OUTPUT_WING : USINT := 5;
	MAX_OUTPUT_CASSETTE : USINT := 1;
	MAX_OUTPUT_EXTERNAL : USINT := 0;
END_VAR
```

#### simFeeder.st
```iecst
ACTION simFeeder:

	IF feeder.activated THEN

		//===============================================================================
		//						Read outputs
		//===============================================================================
		//feeder:this.hw.do_flapOpen
		feeder.hw.out[0].enable := TRUE;
		feeder.hw.out[0].pvName := 'feeder:this.hw.do_flapOpen';
		feeder.hw.out[0]();

		//feeder:this.hw.do_flapClose
		feeder.hw.out[1].enable := TRUE;
		feeder.hw.out[1].pvName := 'feeder:this.hw.do_flapClose';
		feeder.hw.out[1]();

		//feeder:this.hw.do_beltBackwards
		feeder.hw.out[2].enable := TRUE;
		feeder.hw.out[2].pvName := 'feeder:this.hw.do_beltBackwards';
		feeder.hw.out[2]();

		//===============================================================================
		//						Set inputs
		//===============================================================================

		// Set level sensor in bowl high for 5s and low for 10s
		feeder.var.TOF_levelSensorOn(IN := feeder.var.TON_levelSensorOff.Q, PT := T#5s);
		feeder.var.TON_levelSensorOff(IN := NOT feeder.var.TOF_levelSensorOn.Q, PT := T#10s);
		feeder.hw.in[4].setValue := SEL(feeder.var.TOF_levelSensorOn.Q, 0, 1);

		// Set state for flap
		feeder.var.TON_0.PT := T#5s;
		CASE feeder.var.stateFlap OF
			0:
				IF feeder.hw.out[0].actValue = 1 THEN
					feeder.var.stateFlap := 10;
				ELSIF feeder.hw.out[1].actValue = 1 THEN
					feeder.var.stateFlap := 20;
				END_IF
			10:
				feeder.var.TON_0(IN := TRUE);

				IF feeder.var.TON_0.Q THEN
					feeder.var.TON_0(IN := FALSE);
					feeder.hw.in[2].setValue :=	feeder.hw.in[3].setValue := 0;
					feeder.var.stateFlap := 0;
				END_IF
			20:
				feeder.var.TON_0(IN := TRUE);

				IF feeder.var.TON_0.Q THEN
					feeder.var.TON_0(IN := FALSE);
					feeder.hw.in[2].setValue := feeder.hw.in[3].setValue := 1;
					feeder.var.stateFlap := 0;
				END_IF
		END_CASE

		// Set stateFlap for box ready
		feeder.hw.in[1].setValue := feeder.hw.out[2].actValue = 0;

		//::feeder:this.hw.di_levelSensorBelt
		feeder.hw.in[0].enable := TRUE;
		feeder.hw.in[0].dpName := '%IX.IF6.ST9.DigitalInput03';
		feeder.hw.in[0].setValue := 1;
		feeder.hw.in[0]();

		//::feeder:this.hw.di_boxIsReadyAtFlap
		feeder.hw.in[1].enable := TRUE;
		feeder.hw.in[1].dpName := '%IX.IF6.ST9.DigitalInput05';
		feeder.hw.in[1]();

		//::feeder:this.hw.di_flapIsClosed
		feeder.hw.in[2].enable := TRUE;
		feeder.hw.in[2].dpName := '%IX.IF6.ST9.DigitalInput04';
		feeder.hw.in[2]();

		//::feeder:this.hw.di_flapIsOpen
		feeder.hw.in[3].enable := TRUE;
		feeder.hw.in[3].dpName := '%IX.IF6.ST9.DigitalInput02';
		feeder.hw.in[3]();

		//::feeder:this.hw.di_levelSensorInBowl
		feeder.hw.in[4].enable := TRUE;
		feeder.hw.in[4].dpName := '%IX.IF6.ST1.DigitalInput01';
		feeder.hw.in[4]();

	END_IF

END_ACTION
```

#### simVibrator.st
```iecst
ACTION simVibrator:

	FOR i:=0 TO NUM_VIBRATOR DO

		IF vibrator[i].activated THEN

		ELSE

		END_IF

	END_FOR

END_ACTION
```

#### simConveyor.st
```iecst
ACTION simBelt:

	IF belt.activated THEN

		IF belt.usePWMforSim THEN
			// using the PWM

			//===============================================================================
			//						Read outputs
			//===============================================================================
			//this.MTBasicsLimiter_0.Out
			belt.hw.out[0].enable := TRUE;
			belt.hw.out[0].pvName := 'belt:this.MTBasicsLimiter_0.Out';
			belt.hw.out[0]();

			belt.var.convSpeed := UDINT_TO_REAL(belt.hw.out[0].actValue);

			//===============================================================================
			//						Set inputs
			//===============================================================================
			IF belt.hw.in[0].setValue = 0 THEN
				belt.var.TON_sensor.PT := T#300ms;
				belt.var.TON_sensor.IN := SEL(belt.var.convSpeed > 0, FALSE, TRUE);
			ELSE
				belt.var.TON_sensor.PT := T#100ms;
				belt.var.TON_sensor.IN := SEL(belt.var.convSpeed > 0, FALSE, TRUE);
			END_IF

			belt.var.TON_sensor();

			IF belt.var.TON_sensor.Q THEN
				belt.var.TON_sensor.IN := FALSE;
				belt.var.TON_sensor();
				belt.hw.in[0].setValue := SEL(belt.hw.in[0].setValue = 0, 0, 1);
			END_IF

		ELSE
			// using the Servo motor
			//===============================================================================
			//						Read outputs
			//===============================================================================
			//this.MTBasicsLimiter_0.Out
			belt.hw.out[0].enable := TRUE;
			belt.hw.out[0].pvName := 'belt:axis.status.actPosition';
			belt.hw.out[0]();

			belt.var.convPosition := gBeltInterface.status.actualPosition;

			//===============================================================================
			//						Set inputs
			//===============================================================================
			CASE belt.var.state OF
				0:
					belt.var.brickEnd := belt.var.convPosition + belt.var.brickLength;
					IF belt.var.bricksAtEdgeIdx < 300 THEN
						belt.var.bricksAtEdge[belt.var.bricksAtEdgeIdx] := belt.var.brickEnd + 10;
						belt.var.bricksAtEdgeIdx := belt.var.bricksAtEdgeIdx + 1;
					END_IF
					belt.var.brickStart := belt.var.convPosition;
					belt.hw.in[0].setValue := TRUE;
					belt.var.state := 10;

				10:
					IF belt.var.convPosition >= belt.var.brickEnd THEN
						belt.hw.in[0].setValue := FALSE;
						belt.var.gapLength := belt.var.brickLength / ((USINT_TO_REAL(gVibratorInterface[1].status.countingSpeed)/100)*belt.var.percentToSpeed);
						belt.var.gapLengthVarMin := REAL_TO_UDINT(belt.var.gapLength - belt.var.gapLength * belt.var.gapVariancePrc);
						belt.var.gapLengthVarMax := REAL_TO_UDINT(belt.var.gapLength + belt.var.gapLength * belt.var.gapVariancePrc);
						belt.var.brickGap := belt.var.convPosition + UDINT_TO_REAL(rand_interval(belt.var.gapLengthVarMin, belt.var.gapLengthVarMax));
						belt.var.gapStart := belt.var.convPosition;
						belt.var.state := 20;
					ELSIF belt.var.convPosition < belt.var.brickStart THEN
						brsmemset(ADR(belt.var.bricksAtEdge), 0, SIZEOF(belt.var.bricksAtEdge));
						belt.var.bricksAtEdgeIdx := 0;
						brsmemset(ADR(capcon.var.signals), 0, SIZEOF(capcon.var.signals));
						brsmemset(ADR(capcon.var.rejects), 0, SIZEOF(capcon.var.rejects));
						capcon.var.signalIdx := 0;
						belt.var.state := 0;
					END_IF

				20:
					IF belt.var.convPosition >= belt.var.brickGap THEN
						belt.var.state := 0;
					ELSIF belt.var.convPosition < belt.var.gapStart THEN
						brsmemset(ADR(belt.var.bricksAtEdge), 0, SIZEOF(belt.var.bricksAtEdge));
						belt.var.bricksAtEdgeIdx := 0;
						brsmemset(ADR(capcon.var.signals), 0, SIZEOF(capcon.var.signals));
						brsmemset(ADR(capcon.var.rejects), 0, SIZEOF(capcon.var.rejects));
						capcon.var.signalIdx := 0;
						belt.var.state := 0;
					END_IF
			END_CASE

			gSimulation.status.photoSensor := belt.hw.in[0].setValue = 1;

//			IF (REAL_TO_UDINT(belt.var.convPosition) MOD 400) > 370 THEN
//				belt.hw.in[0].setValue := TRUE;
//			ELSE
//				belt.hw.in[0].setValue := FALSE;
//			END_IF

		END_IF
	END_IF

END_ACTION
```

#### simCapcon.st
```iecst
ACTION simCapcon:

	IF capcon.activated THEN

		//===============================================================================
		//						Set inputs
		//===============================================================================

		capcon.var.beltPosition := gBeltInterface.status.actualPosition;

		IF capcon.var.beltPosition > belt.var.bricksAtEdge[0] AND belt.var.bricksAtEdgeIdx > 0 THEN
			capcon.var.signals[capcon.var.signalIdx] := 0;
			capcon.var.rejects[capcon.var.signalIdx] := random() < REAL_TO_INT(65534*(capcon.var.errorRate/100)-32767);
			capcon.var.signalIdx := capcon.var.signalIdx + 1;
			IF belt.var.bricksAtEdgeIdx > 0 THEN
				FOR capcon.var.i:=1 TO belt.var.bricksAtEdgeIdx DO
					belt.var.bricksAtEdge[capcon.var.i-1] := belt.var.bricksAtEdge[capcon.var.i];
				END_FOR
				belt.var.bricksAtEdgeIdx := belt.var.bricksAtEdgeIdx - 1;
			END_IF
		END_IF

		capcon.var.currSignal := 0;
		IF capcon.var.signalIdx > 0 THEN
			FOR capcon.var.i:=0 TO capcon.var.signalIdx-1 DO
				IF capcon.var.signals[capcon.var.i] > 50 THEN
					capcon.var.x := (capcon.var.signals[capcon.var.i]-97)/4.6;
					IF capcon.var.x = 0 THEN
						capcon.var.x := 0.001;
					END_IF
					capcon.var.currSignal := capcon.var.currSignal + (SIN(capcon.var.x)*SEL(capcon.var.rejects[capcon.var.i], capcon.var.signalHeight, capcon.var.signalHeight*3)/capcon.var.x) * (1/SQRT(2*amPI*pow(0.3, 2))) * EXP((-pow(capcon.var.x-0, 2))/2*pow(0.3, 2));
				END_IF
				capcon.var.signals[capcon.var.i] := capcon.var.signals[capcon.var.i] + 1;
			END_FOR
			IF capcon.var.signals[0] > 143 THEN
				FOR capcon.var.i:=1 TO capcon.var.signalIdx DO
					capcon.var.signals[capcon.var.i-1] := capcon.var.signals[capcon.var.i];
					capcon.var.rejects[capcon.var.i-1] := capcon.var.rejects[capcon.var.i];
				END_FOR
				capcon.var.signalIdx := capcon.var.signalIdx - 1;
			END_IF
		END_IF

		gSimCapcon.status.simSignal := REAL_TO_INT(capcon.var.currSignal);
	END_IF

END_ACTION
```
